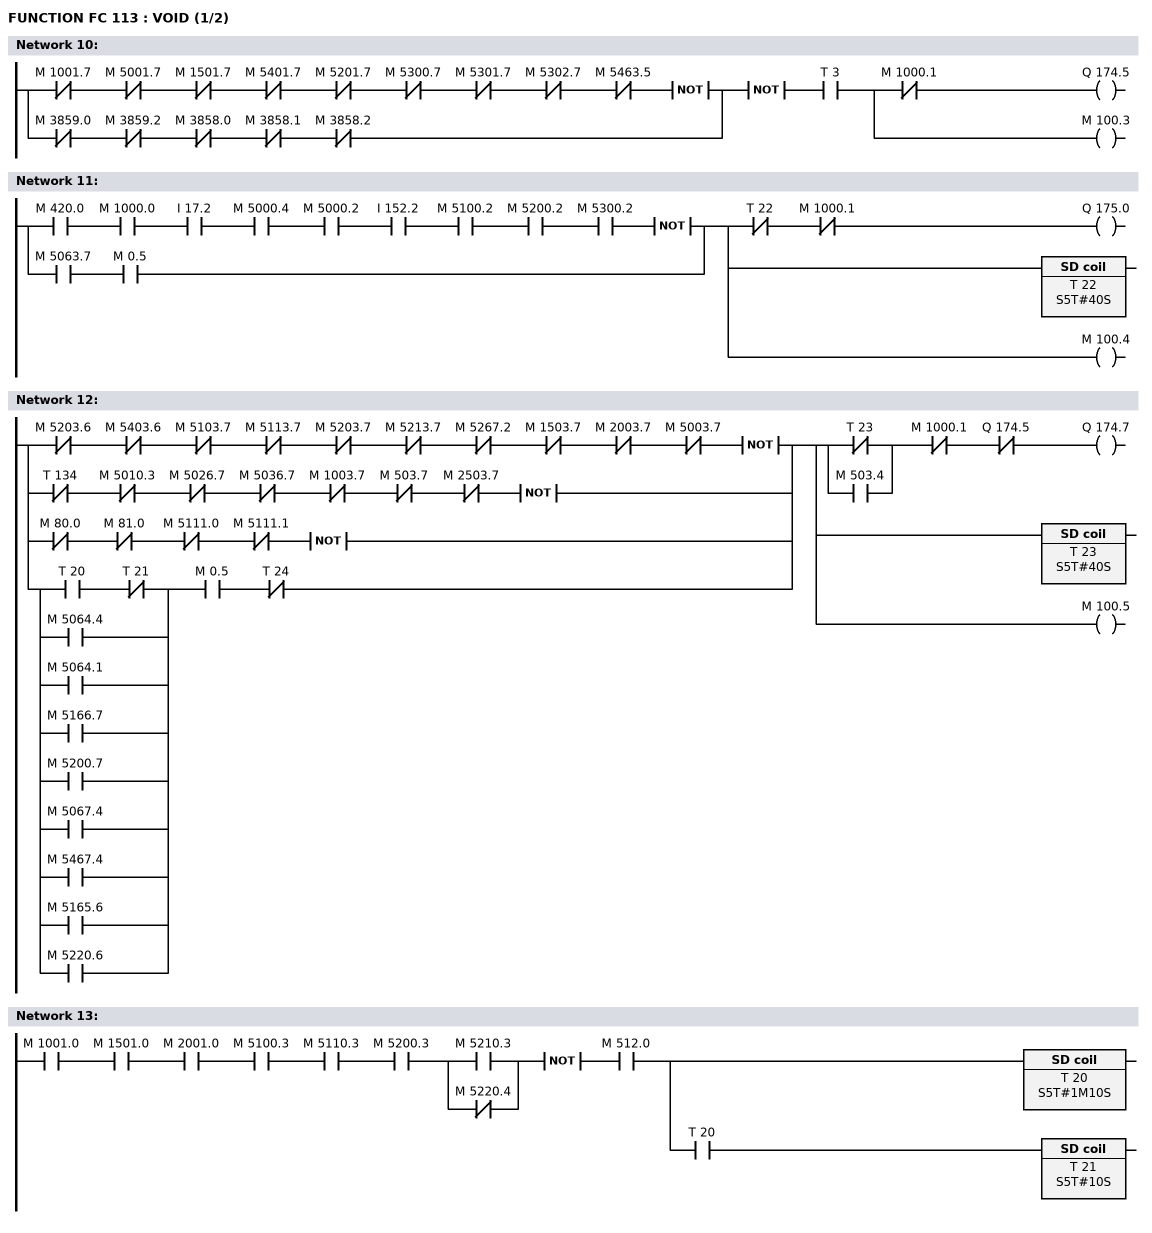

      AN    M   1001.7;
      AN    M   5001.7;
      AN    M   1501.7;
      AN    M   5401.7;
      AN    M   5201.7;
      AN    M   5300.7;
      AN    M   5301.7;
      AN    M   5302.7;
      AN    M   5463.5;
      NOT   ;
      O     ;
      AN    M   3859.0;
      AN    M   3859.2;
      AN    M   3858.0;
      AN    M   3858.1;
      AN    M   3858.2;
      NOT   ;
      A     T      3;
      =     L      0.0;
      A     L      0.0;
      AN    M   1000.1;
      =     Q    174.5;
      A     L      0.0;
      BLD   102;
      =     M    100.3;
NETWORK
TITLE =

      A     M    420.0;
      A     M   1000.0;
      A     I     17.2;
      A     M   5000.4;
      A     M   5000.2;
      A     I    152.2;
      A     M   5100.2;
      A     M   5200.2;
      A     M   5300.2;
      NOT   ;
      O     ;
      A     M   5063.7;
      A     M      0.5;
      =     L      0.0;
      A     L      0.0;
      AN    T     22;
      AN    M   1000.1;
      =     Q    175.0;
      A     L      0.0;
      BLD   102;
      L     S5T#40S;
      SD    T     22;
      A     L      0.0;
      BLD   102;
      =     M    100.4;
NETWORK
TITLE =

      AN    M   5203.6;
      AN    M   5403.6;
      AN    M   5103.7;
      AN    M   5113.7;
      AN    M   5203.7;
      AN    M   5213.7;
      AN    M   5267.2;
      AN    M   1503.7;
      AN    M   2003.7;
      AN    M   5003.7;
      NOT   ;
      O(    ;
      AN    T    134;
      AN    M   5010.3;
      AN    M   5026.7;
      AN    M   5036.7;
      AN    M   1003.7;
      AN    M    503.7;
      AN    M   2503.7;
      NOT   ;
      )     ;
      O(    ;
      AN    M     80.0;
      AN    M     81.0;
      AN    M   5111.0;
      AN    M   5111.1;
      NOT   ;
      )     ;
      O     ;
      A(    ;
      A     T     20;
      AN    T     21;
      O     M   5064.4;
      O     M   5064.1;
      O     M   5166.7;
      O     M   5200.7;
      O     M   5067.4;
      O     M   5467.4;
      O     M   5165.6;
      O     M   5220.6;
      )     ;
      A     M      0.5;
      AN    T     24;
      =     L      0.0;
      A     L      0.0;
      A(    ;
      ON    T     23;
      O     M    503.4;
      )     ;
      AN    M   1000.1;
      AN    Q    174.5;
      =     Q    174.7;
      A     L      0.0;
      BLD   102;
      L     S5T#40S;
      SD    T     23;
      A     L      0.0;
      BLD   102;
      =     M    100.5;
NETWORK
TITLE =

      A     M   1001.0;
      A     M   1501.0;
      A     M   2001.0;
      A     M   5100.3;
      A     M   5110.3;
      A     M   5200.3;
      A(    ;
      O     M   5210.3;
      ON    M   5220.4;
      )     ;
      NOT   ;
      A     M    512.0;
      =     L      0.0;
      A     L      0.0;
      BLD   102;
      L     S5T#1M10S;
      SD    T     20;
      A     L      0.0;
      A     T     20;
      L     S5T#10S;
      SD    T     21;
NETWORK
TITLE =
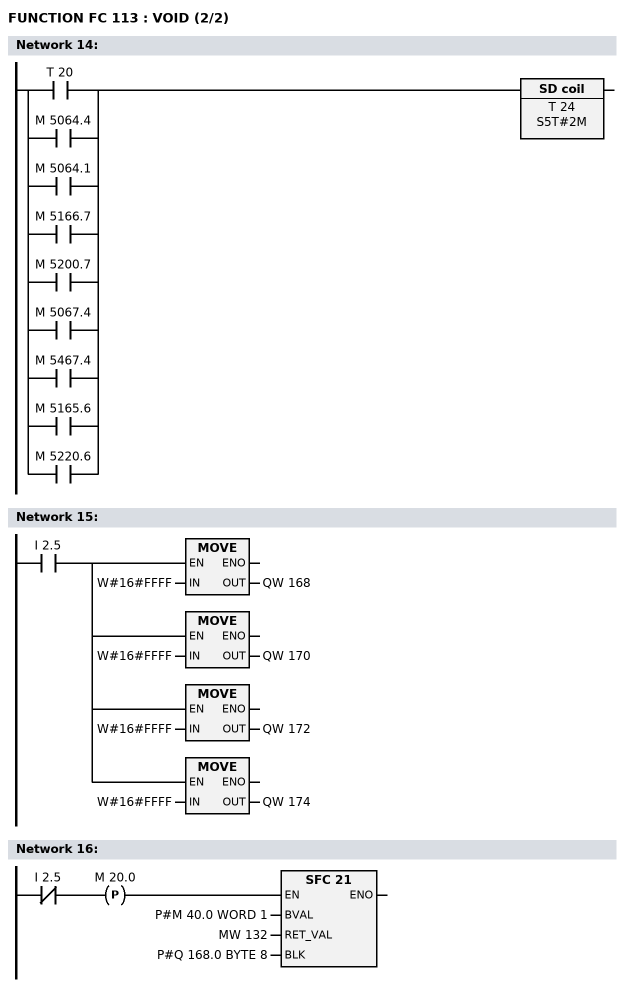

      O     T     20;
      O     M   5064.4;
      O     M   5064.1;
      O     M   5166.7;
      O     M   5200.7;
      O     M   5067.4;
      O     M   5467.4;
      O     M   5165.6;
      O     M   5220.6;
      L     S5T#2M;
      SD    T     24;
NETWORK
TITLE =

      A     I      2.5;
      =     L      0.0;
      A     L      0.0;
      JNB   _003;
      L     W#16#FFFF;
      T     QW   168;
_003: NOP   0;
      A     L      0.0;
      JNB   _004;
      L     W#16#FFFF;
      T     QW   170;
_004: NOP   0;
      A     L      0.0;
      JNB   _005;
      L     W#16#FFFF;
      T     QW   172;
_005: NOP   0;
      A     L      0.0;
      JNB   _006;
      L     W#16#FFFF;
      T     QW   174;
_006: NOP   0;
NETWORK
TITLE =

      AN    I      2.5;
      FP    M     20.0;
      JNB   _007;
      CALL SFC   21 (
           BVAL                     := P#M 40.0 WORD 1,
           RET_VAL                  := MW   132,
           BLK                      := P#Q 168.0 BYTE 8);
_007: NOP   0;
END_FUNCTION

FUNCTION_BLOCK FB 120
TITLE =
VERSION : 0.1


VAR
  S702_MODE : FB 402;
END_VAR
BEGIN
NETWORK
TITLE =
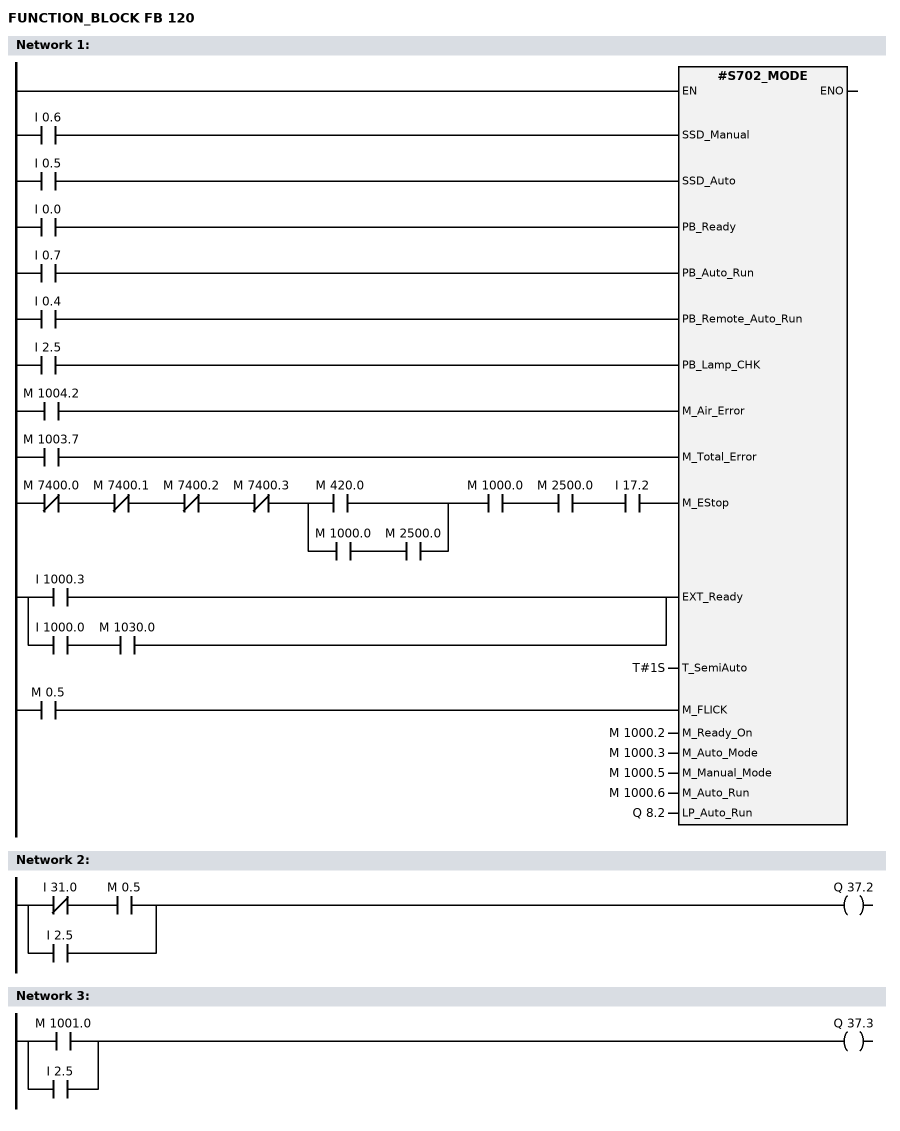

      A     I      0.6;
      =     L      0.0;
      BLD   103;
      A     I      0.5;
      =     L      0.1;
      BLD   103;
      A     I      0.0;
      =     L      0.2;
      BLD   103;
      A     I      0.7;
      =     L      0.3;
      BLD   103;
      A     I      0.4;
      =     L      0.5;
      BLD   103;
      A     I      2.5;
      =     L      0.6;
      BLD   103;
      A     M   1004.2;
      =     L      0.7;
      BLD   103;
      A     M   1003.7;
      =     L      1.1;
      BLD   103;
      AN    M   7400.0;
      AN    M   7400.1;
      AN    M   7400.2;
      AN    M   7400.3;
      A(    ;
      O     M    420.0;
      O     ;
      A     M   1000.0;
      A     M   2500.0;
      )     ;
      A     M   1000.0;
      A     M   2500.0;
      A     I     17.2;
      =     L      1.2;
      BLD   103;
      A(    ;
      O     I   1000.3;
      O     ;
      A     I   1000.0;
      A     M   1030.0;
      )     ;
      =     L      1.3;
      BLD   103;
      A     M      0.5;
      =     L      1.5;
      BLD   103;
      CALL #S702_MODE (
           SSD_Manual               := L      0.0,
           SSD_Auto                 := L      0.1,
           PB_Ready                 := L      0.2,
           PB_Auto_Run              := L      0.3,
           PB_Remote_Auto_Run       := L      0.5,
           PB_Lamp_CHK              := L      0.6,
           M_Air_Error              := L      0.7,
           M_Total_Error            := L      1.1,
           M_EStop                  := L      1.2,
           EXT_Ready                := L      1.3,
           T_SemiAuto               := T#1S,
           M_FLICK                  := L      1.5,
           M_Ready_On               := M   1000.2,
           M_Auto_Mode              := M   1000.3,
           M_Manual_Mode            := M   1000.5,
           M_Auto_Run               := M   1000.6,
           LP_Auto_Run              := Q      8.2);
      NOP   0;
NETWORK
TITLE =

      AN    I     31.0;
      A     M      0.5;
      O     I      2.5;
      =     Q     37.2;
NETWORK
TITLE =

      O     M   1001.0;
      O     I      2.5;
      =     Q     37.3;
END_FUNCTION_BLOCK

DATA_BLOCK DB 120
TITLE =
VERSION : 0.0

 FB 120
BEGIN
   S702_MODE.SSD_Manual := FALSE;
   S702_MODE.SSD_Auto := FALSE;
   S702_MODE.PB_Ready := FALSE;
   S702_MODE.PB_Auto_Run := FALSE;
   S702_MODE.PB_Remote_Ready := FALSE;
   S702_MODE.PB_Remote_Auto_Run := FALSE;
   S702_MODE.PB_Lamp_CHK := FALSE;
   S702_MODE.M_Air_Error := FALSE;
   S702_MODE.M_Water_Error := FALSE;
   S702_MODE.M_Total_Error := FALSE;
   S702_MODE.M_EStop := FALSE;
   S702_MODE.EXT_Ready := FALSE;
   S702_MODE.EXT_Auto := FALSE;
   S702_MODE.T_SemiAuto := T#0MS;
   S702_MODE.M_FLICK := FALSE;
   S702_MODE.M_Ready_On := FALSE;
   S702_MODE.M_Auto_Mode := FALSE;
   S702_MODE.M_SemiAuto_Mode := FALSE;
   S702_MODE.M_Manual_Mode := FALSE;
   S702_MODE.M_Auto_Run := FALSE;
   S702_MODE.LP_Ready_On := FALSE;
   S702_MODE.LP_Auto_Run := FALSE;
   S702_MODE.AUTO_MODE_DELAY.IN := FALSE;
   S702_MODE.AUTO_MODE_DELAY.PT := T#0MS;
   S702_MODE.AUTO_MODE_DELAY.Q := FALSE;
   S702_MODE.AUTO_MODE_DELAY.ET := T#0MS;
   S702_MODE.AUTO_MODE_DELAY.STATE := B#16#0;
   S702_MODE.AUTO_MODE_DELAY.STIME := T#0MS;
   S702_MODE.AUTO_MODE_DELAY.ATIME := T#0MS;
   S702_MODE.SEMI_AUTO_DELAY.IN := FALSE;
   S702_MODE.SEMI_AUTO_DELAY.PT := T#0MS;
   S702_MODE.SEMI_AUTO_DELAY.Q := FALSE;
   S702_MODE.SEMI_AUTO_DELAY.ET := T#0MS;
   S702_MODE.SEMI_AUTO_DELAY.STATE := B#16#0;
   S702_MODE.SEMI_AUTO_DELAY.STIME := T#0MS;
   S702_MODE.SEMI_AUTO_DELAY.ATIME := T#0MS;
   S702_MODE.MANUAL_DELAY.IN := FALSE;
   S702_MODE.MANUAL_DELAY.PT := T#0MS;
   S702_MODE.MANUAL_DELAY.Q := FALSE;
   S702_MODE.MANUAL_DELAY.ET := T#0MS;
   S702_MODE.MANUAL_DELAY.STATE := B#16#0;
   S702_MODE.MANUAL_DELAY.STIME := T#0MS;
   S702_MODE.MANUAL_DELAY.ATIME := T#0MS;
END_DATA_BLOCK

FUNCTION FC 120 : VOID
TITLE =
VERSION : 0.1

BEGIN
NETWORK
TITLE =
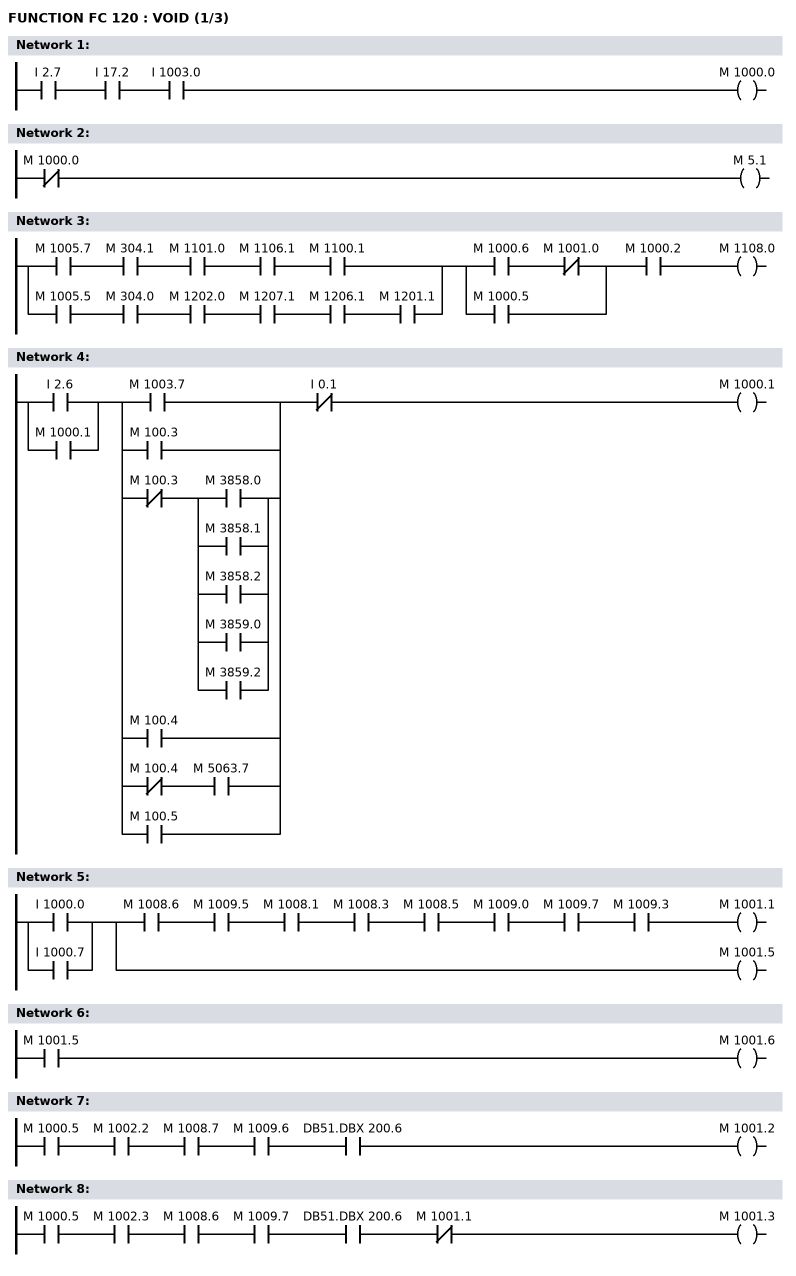

      A     I      2.7;
      A     I     17.2;
      A     I   1003.0;
      =     M   1000.0;
NETWORK
TITLE =

      AN    M   1000.0;
      =     M      5.1;
NETWORK
TITLE =

      A(    ;
      A     M   1005.7;
      A     M    304.1;
      A     M   1101.0;
      A     M   1106.1;
      A     M   1100.1;
      O     ;
      A     M   1005.5;
      A     M    304.0;
      A     M   1202.0;
      A     M   1207.1;
      A     M   1206.1;
      A     M   1201.1;
      )     ;
      A(    ;
      A     M   1000.6;
      AN    M   1001.0;
      O     M   1000.5;
      )     ;
      A     M   1000.2;
      =     M   1108.0;
NETWORK
TITLE =

      A(    ;
      O     I      2.6;
      O     M   1000.1;
      )     ;
      A(    ;
      O     M   1003.7;
      O     M    100.3;
      O     ;
      AN    M    100.3;
      A(    ;
      O     M   3858.0;
      O     M   3858.1;
      O     M   3858.2;
      O     M   3859.0;
      O     M   3859.2;
      )     ;
      O     M    100.4;
      O     ;
      AN    M    100.4;
      A     M   5063.7;
      O     M    100.5;
      )     ;
      AN    I      0.1;
      =     M   1000.1;
NETWORK
TITLE =

      O     I   1000.0;
      O     I   1000.7;
      =     L      0.0;
      A     L      0.0;
      A     M   1008.6;
      A     M   1009.5;
      A     M   1008.1;
      A     M   1008.3;
      A     M   1008.5;
      A     M   1009.0;
      A     M   1009.7;
      A     M   1009.3;
      =     M   1001.1;
      A     L      0.0;
      BLD   102;
      =     M   1001.5;
NETWORK
TITLE =

      A     M   1001.5;
      =     M   1001.6;
NETWORK
TITLE =

      A     M   1000.5;
      A     M   1002.2;
      A     M   1008.7;
      A     M   1009.6;
      A     DB51.DBX  200.6;
      =     M   1001.2;
NETWORK
TITLE =

      A     M   1000.5;
      A     M   1002.3;
      A     M   1008.6;
      A     M   1009.7;
      A     DB51.DBX  200.6;
      AN    M   1001.1;
      =     M   1001.3;
NETWORK
TITLE =
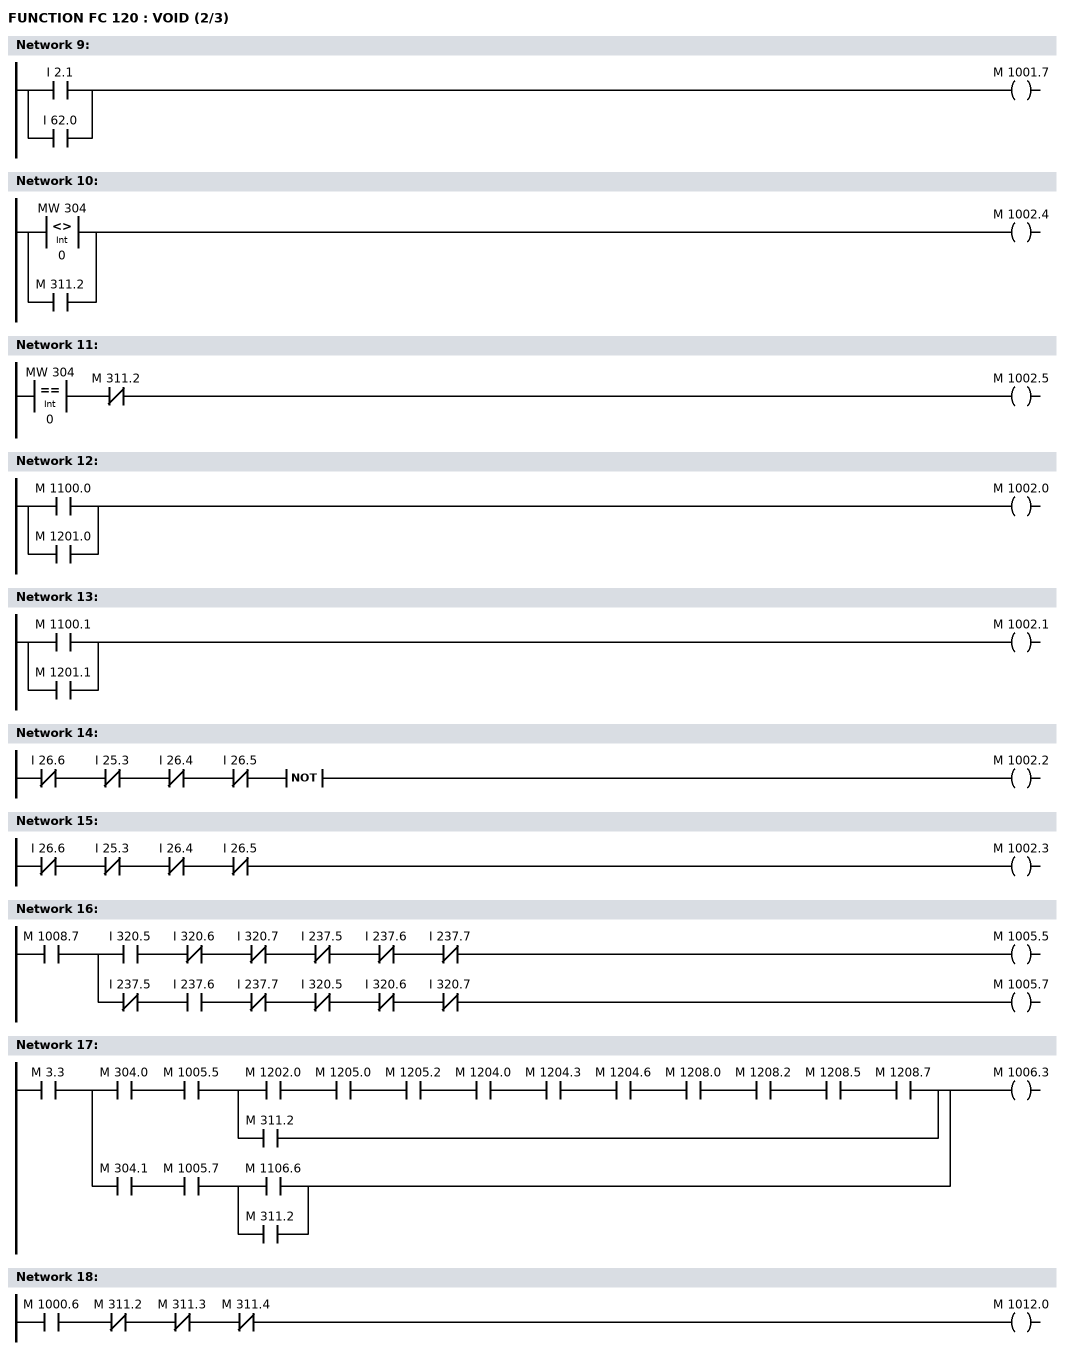

      O     I      2.1;
      O     I     62.0;
      =     M   1001.7;
NETWORK
TITLE =

      O(    ;
      L     MW   304;
      L     0;
      <>I   ;
      )     ;
      O     M    311.2;
      =     M   1002.4;
NETWORK
TITLE =

      A(    ;
      L     MW   304;
      L     0;
      ==I   ;
      )     ;
      AN    M    311.2;
      =     M   1002.5;
NETWORK
TITLE =

      O     M   1100.0;
      O     M   1201.0;
      =     M   1002.0;
NETWORK
TITLE =

      O     M   1100.1;
      O     M   1201.1;
      =     M   1002.1;
NETWORK
TITLE =

      AN    I     26.6;
      AN    I     25.3;
      AN    I     26.4;
      AN    I     26.5;
      NOT   ;
      =     M   1002.2;
NETWORK
TITLE =

      AN    I     26.6;
      AN    I     25.3;
      AN    I     26.4;
      AN    I     26.5;
      =     M   1002.3;
NETWORK
TITLE =

      A     M   1008.7;
      =     L      0.0;
      A     L      0.0;
      A     I    320.5;
      AN    I    320.6;
      AN    I    320.7;
      AN    I    237.5;
      AN    I    237.6;
      AN    I    237.7;
      =     M   1005.5;
      A     L      0.0;
      AN    I    237.5;
      A     I    237.6;
      AN    I    237.7;
      AN    I    320.5;
      AN    I    320.6;
      AN    I    320.7;
      =     M   1005.7;
NETWORK
TITLE =

      A     M      3.3;
      A(    ;
      A     M    304.0;
      A     M   1005.5;
      A(    ;
      A     M   1202.0;
      A     M   1205.0;
      A     M   1205.2;
      A     M   1204.0;
      A     M   1204.3;
      A     M   1204.6;
      A     M   1208.0;
      A     M   1208.2;
      A     M   1208.5;
      A     M   1208.7;
      O     M    311.2;
      )     ;
      O     ;
      A     M    304.1;
      A     M   1005.7;
      A(    ;
      O     M   1106.6;
      O     M    311.2;
      )     ;
      )     ;
      =     M   1006.3;
NETWORK
TITLE =

      A     M   1000.6;
      AN    M    311.2;
      AN    M    311.3;
      AN    M    311.4;
      =     M   1012.0;
NETWORK
TITLE =
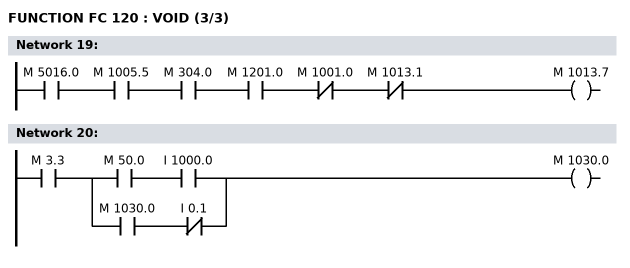

      A     M   5016.0;
      A     M   1005.5;
      A     M    304.0;
      A     M   1201.0;
      AN    M   1001.0;
      AN    M   1013.1;
      =     M   1013.7;
NETWORK
TITLE =

      A     M      3.3;
      A(    ;
      A     M     50.0;
      A     I   1000.0;
      O     ;
      A     M   1030.0;
      AN    I      0.1;
      )     ;
      =     M   1030.0;
NETWORK
TITLE =

      AN    OV;
      =     L      0.0;
      A(    ;
      A(    ;
      A     L      0.0;
      AN    M   1005.7;
      JNB   _001;
      L     0;
      T     MW  1150;
      SET   ;
      SAVE  ;
      CLR   ;
_001: A     BR;
      )     ;
      JNB   _002;
      L     0;
      T     MW  1152;
      SET   ;
      SAVE  ;
      CLR   ;
_002: A     BR;
      )     ;
      JNB   _003;
      L     0;
      T     MB  1154;
_003: NOP   0;
      A(    ;
      A(    ;
      A     L      0.0;
      AN    M   1005.5;
      JNB   _004;
      L     0;
      T     MW  1250;
      SET   ;
      SAVE  ;
      CLR   ;
_004: A     BR;
      )     ;
      JNB   _005;
      L     0;
      T     MW  1252;
      SET   ;
      SAVE  ;
      CLR   ;
_005: A     BR;
      )     ;
      JNB   _006;
      L     0;
      T     MB  1254;
_006: NOP   0;
NETWORK
TITLE =

      AN    M   1007.4;
      =     L      0.0;
      A     L      0.0;
      JNB   _007;
      CALL SFC   21 (
           BVAL                     := P#M 40.0 WORD 1,
           RET_VAL                  := MW   132,
           BLK                      := P#M 1100.0 BYTE 10);
_007: NOP   0;
      A     L      0.0;
      JNB   _008;
      CALL SFC   21 (
           BVAL                     := P#M 40.0 WORD 1,
           RET_VAL                  := MW   132,
           BLK                      := P#Q 236.0 BYTE 4);
_008: NOP   0;
      A     L      0.0;
      JNB   _009;
      CALL SFC   21 (
           BVAL                     := P#M 40.0 WORD 1,
           RET_VAL                  := MW   132,
           BLK                      := P#M 1200.0 BYTE 12);
_009: NOP   0;
      A     L      0.0;
      JNB   _00a;
      CALL SFC   21 (
           BVAL                     := P#M 40.0 WORD 1,
           RET_VAL                  := MW   132,
           BLK                      := P#M 1240.0 BYTE 5);
_00a: NOP   0;
      A     L      0.0;
      JNB   _00b;
      CALL SFC   21 (
           BVAL                     := P#M 40.0 WORD 1,
           RET_VAL                  := MW   132,
           BLK                      := P#Q 332.0 BYTE 6);
_00b: NOP   0;
END_FUNCTION

FUNCTION_BLOCK FB 121
TITLE =
VERSION : 0.1


VAR
  S702_HOOK_PIN : FB 424;
  S702_DAECHA_LOCK : FB 424;
  S702_DAECHA_LOCK_UP_DN : FB 424;
  S702_ELE : FB 424;
  S702_AIR_ELE : FB 424;
  S702_EJECT : FB 424;
  S702_DAECHA_STOPPER : FB 424;
  S702_DAECHA_CLAMP : FB 424;
  S702_SHOCK_ABSORBER : FB 424;
END_VAR
BEGIN
NETWORK
TITLE =
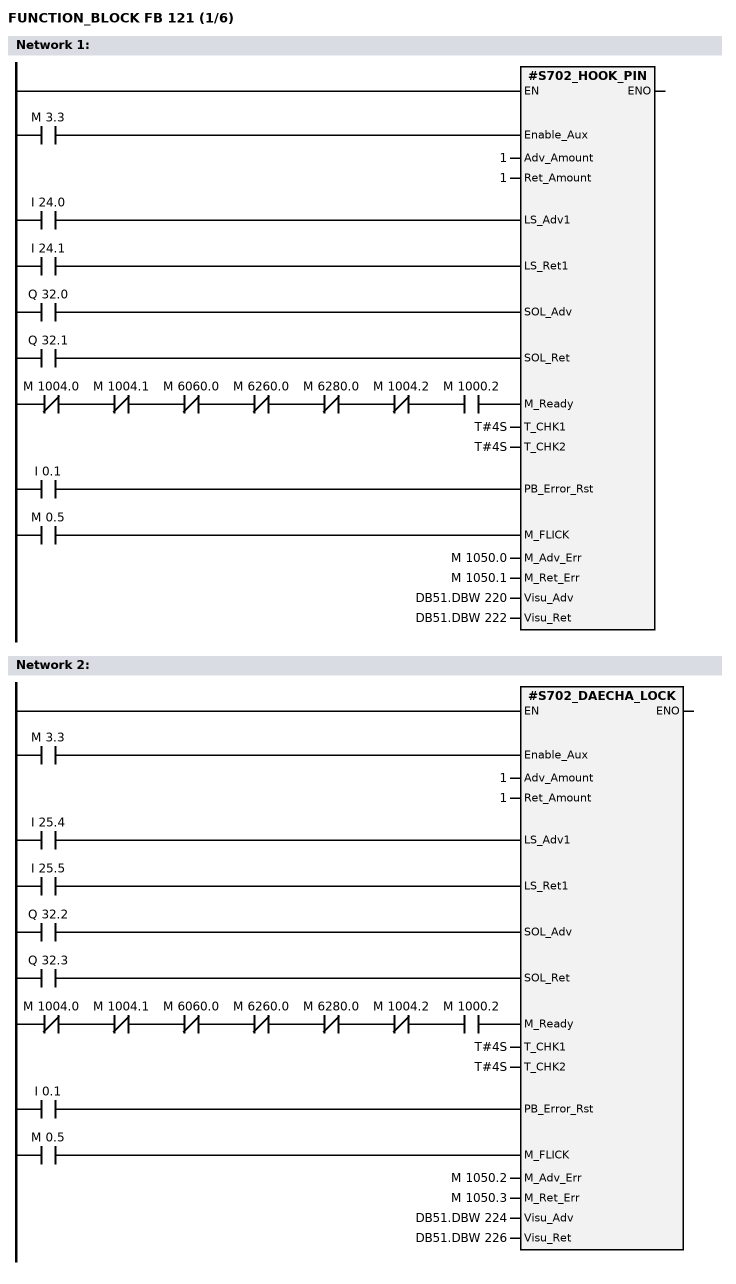

      A     M      3.3;
      =     L      0.0;
      BLD   103;
      A     I     24.0;
      =     L      0.1;
      BLD   103;
      A     I     24.1;
      =     L      0.2;
      BLD   103;
      A     Q     32.0;
      =     L      1.1;
      BLD   103;
      A     Q     32.1;
      =     L      1.2;
      BLD   103;
      AN    M   1004.0;
      AN    M   1004.1;
      AN    M   6060.0;
      AN    M   6260.0;
      AN    M   6280.0;
      AN    M   1004.2;
      A     M   1000.2;
      =     L      1.3;
      BLD   103;
      A     I      0.1;
      =     L      1.5;
      BLD   103;
      A     M      0.5;
      =     L      1.6;
      BLD   103;
      CALL #S702_HOOK_PIN (
           Enable_Aux               := L      0.0,
           Adv_Amount               := 1,
           Ret_Amount               := 1,
           LS_Adv1                  := L      0.1,
           LS_Ret1                  := L      0.2,
           SOL_Adv                  := L      1.1,
           SOL_Ret                  := L      1.2,
           M_Ready                  := L      1.3,
           T_CHK1                   := T#4S,
           T_CHK2                   := T#4S,
           PB_Error_Rst             := L      1.5,
           M_FLICK                  := L      1.6,
           M_Adv_Err                := M   1050.0,
           M_Ret_Err                := M   1050.1,
           Visu_Adv                 := DB51.DBW  220,
           Visu_Ret                 := DB51.DBW  222);
      NOP   0;
NETWORK
TITLE =

      A     M      3.3;
      =     L      0.0;
      BLD   103;
      A     I     25.4;
      =     L      0.1;
      BLD   103;
      A     I     25.5;
      =     L      0.2;
      BLD   103;
      A     Q     32.2;
      =     L      1.1;
      BLD   103;
      A     Q     32.3;
      =     L      1.2;
      BLD   103;
      AN    M   1004.0;
      AN    M   1004.1;
      AN    M   6060.0;
      AN    M   6260.0;
      AN    M   6280.0;
      AN    M   1004.2;
      A     M   1000.2;
      =     L      1.3;
      BLD   103;
      A     I      0.1;
      =     L      1.5;
      BLD   103;
      A     M      0.5;
      =     L      1.6;
      BLD   103;
      CALL #S702_DAECHA_LOCK (
           Enable_Aux               := L      0.0,
           Adv_Amount               := 1,
           Ret_Amount               := 1,
           LS_Adv1                  := L      0.1,
           LS_Ret1                  := L      0.2,
           SOL_Adv                  := L      1.1,
           SOL_Ret                  := L      1.2,
           M_Ready                  := L      1.3,
           T_CHK1                   := T#4S,
           T_CHK2                   := T#4S,
           PB_Error_Rst             := L      1.5,
           M_FLICK                  := L      1.6,
           M_Adv_Err                := M   1050.2,
           M_Ret_Err                := M   1050.3,
           Visu_Adv                 := DB51.DBW  224,
           Visu_Ret                 := DB51.DBW  226);
      NOP   0;
NETWORK
TITLE =
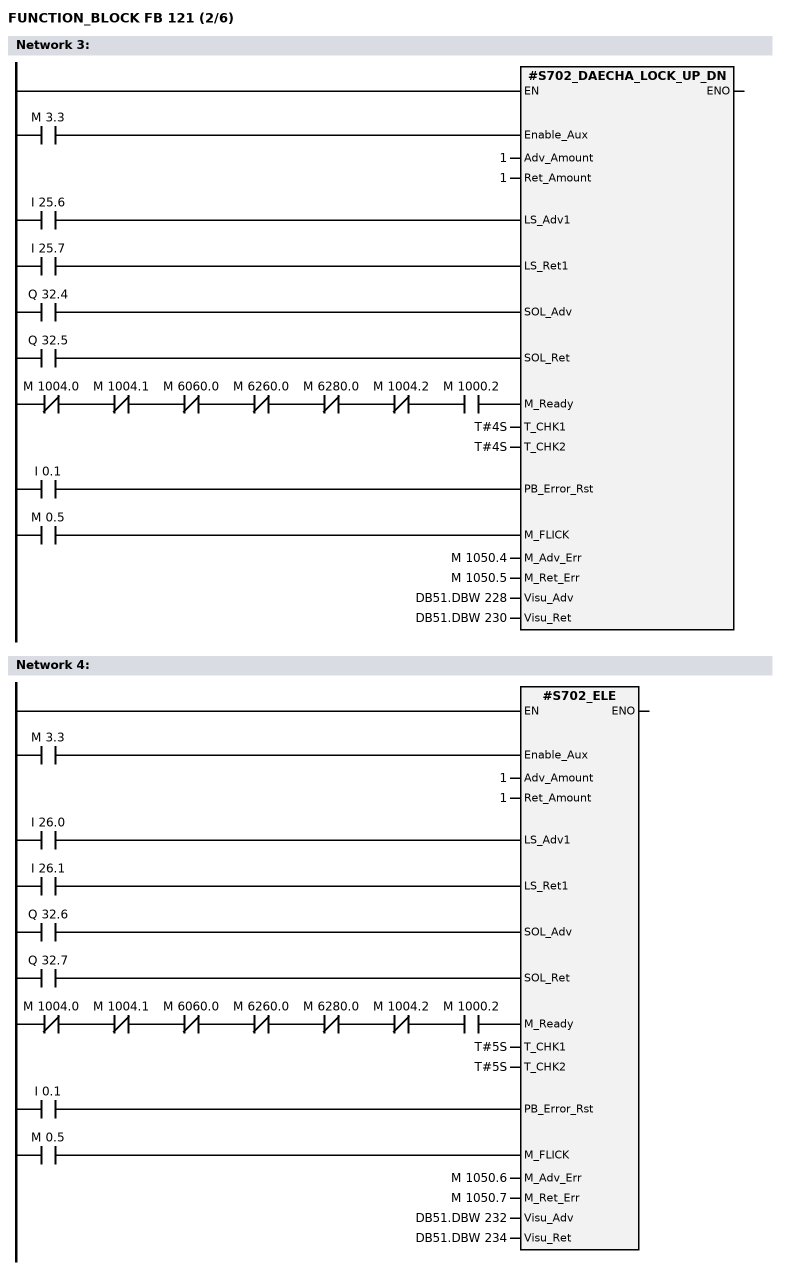

      A     M      3.3;
      =     L      0.0;
      BLD   103;
      A     I     25.6;
      =     L      0.1;
      BLD   103;
      A     I     25.7;
      =     L      0.2;
      BLD   103;
      A     Q     32.4;
      =     L      1.1;
      BLD   103;
      A     Q     32.5;
      =     L      1.2;
      BLD   103;
      AN    M   1004.0;
      AN    M   1004.1;
      AN    M   6060.0;
      AN    M   6260.0;
      AN    M   6280.0;
      AN    M   1004.2;
      A     M   1000.2;
      =     L      1.3;
      BLD   103;
      A     I      0.1;
      =     L      1.5;
      BLD   103;
      A     M      0.5;
      =     L      1.6;
      BLD   103;
      CALL #S702_DAECHA_LOCK_UP_DN (
           Enable_Aux               := L      0.0,
           Adv_Amount               := 1,
           Ret_Amount               := 1,
           LS_Adv1                  := L      0.1,
           LS_Ret1                  := L      0.2,
           SOL_Adv                  := L      1.1,
           SOL_Ret                  := L      1.2,
           M_Ready                  := L      1.3,
           T_CHK1                   := T#4S,
           T_CHK2                   := T#4S,
           PB_Error_Rst             := L      1.5,
           M_FLICK                  := L      1.6,
           M_Adv_Err                := M   1050.4,
           M_Ret_Err                := M   1050.5,
           Visu_Adv                 := DB51.DBW  228,
           Visu_Ret                 := DB51.DBW  230);
      NOP   0;
NETWORK
TITLE =

      A     M      3.3;
      =     L      0.0;
      BLD   103;
      A     I     26.0;
      =     L      0.1;
      BLD   103;
      A     I     26.1;
      =     L      0.2;
      BLD   103;
      A     Q     32.6;
      =     L      1.1;
      BLD   103;
      A     Q     32.7;
      =     L      1.2;
      BLD   103;
      AN    M   1004.0;
      AN    M   1004.1;
      AN    M   6060.0;
      AN    M   6260.0;
      AN    M   6280.0;
      AN    M   1004.2;
      A     M   1000.2;
      =     L      1.3;
      BLD   103;
      A     I      0.1;
      =     L      1.5;
      BLD   103;
      A     M      0.5;
      =     L      1.6;
      BLD   103;
      CALL #S702_ELE (
           Enable_Aux               := L      0.0,
           Adv_Amount               := 1,
           Ret_Amount               := 1,
           LS_Adv1                  := L      0.1,
           LS_Ret1                  := L      0.2,
           SOL_Adv                  := L      1.1,
           SOL_Ret                  := L      1.2,
           M_Ready                  := L      1.3,
           T_CHK1                   := T#5S,
           T_CHK2                   := T#5S,
           PB_Error_Rst             := L      1.5,
           M_FLICK                  := L      1.6,
           M_Adv_Err                := M   1050.6,
           M_Ret_Err                := M   1050.7,
           Visu_Adv                 := DB51.DBW  232,
           Visu_Ret                 := DB51.DBW  234);
      NOP   0;
NETWORK
TITLE =
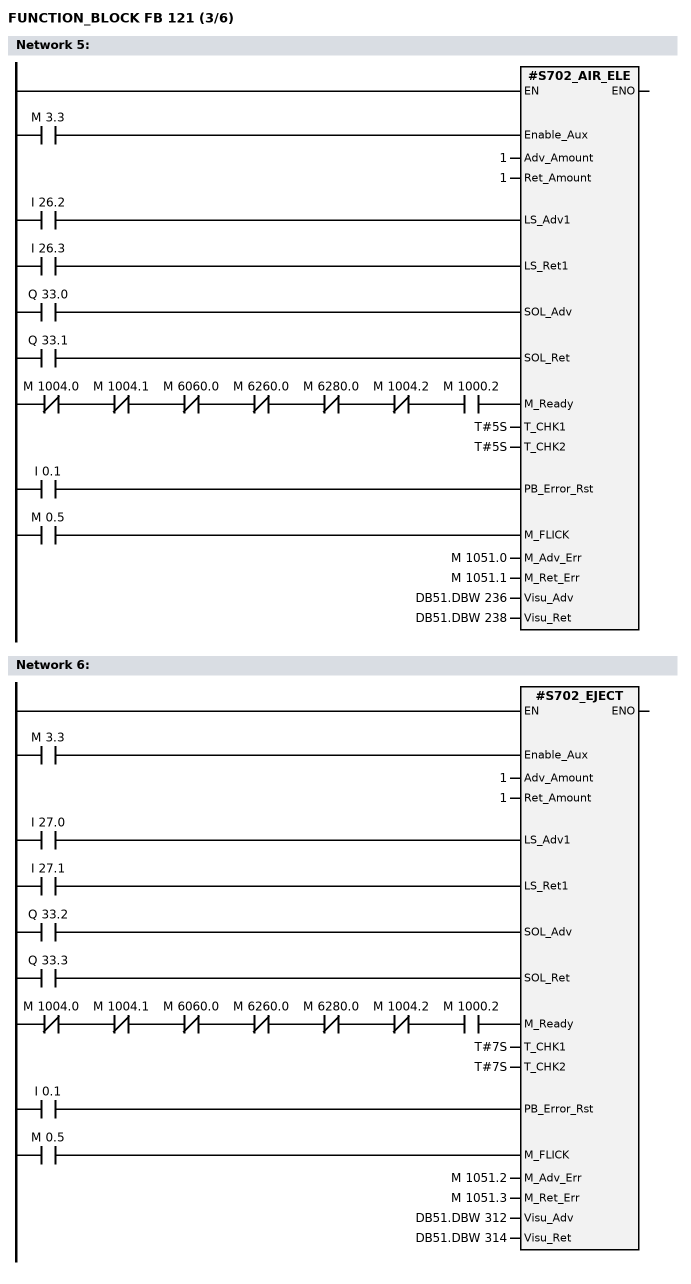

      A     M      3.3;
      =     L      0.0;
      BLD   103;
      A     I     26.2;
      =     L      0.1;
      BLD   103;
      A     I     26.3;
      =     L      0.2;
      BLD   103;
      A     Q     33.0;
      =     L      1.1;
      BLD   103;
      A     Q     33.1;
      =     L      1.2;
      BLD   103;
      AN    M   1004.0;
      AN    M   1004.1;
      AN    M   6060.0;
      AN    M   6260.0;
      AN    M   6280.0;
      AN    M   1004.2;
      A     M   1000.2;
      =     L      1.3;
      BLD   103;
      A     I      0.1;
      =     L      1.5;
      BLD   103;
      A     M      0.5;
      =     L      1.6;
      BLD   103;
      CALL #S702_AIR_ELE (
           Enable_Aux               := L      0.0,
           Adv_Amount               := 1,
           Ret_Amount               := 1,
           LS_Adv1                  := L      0.1,
           LS_Ret1                  := L      0.2,
           SOL_Adv                  := L      1.1,
           SOL_Ret                  := L      1.2,
           M_Ready                  := L      1.3,
           T_CHK1                   := T#5S,
           T_CHK2                   := T#5S,
           PB_Error_Rst             := L      1.5,
           M_FLICK                  := L      1.6,
           M_Adv_Err                := M   1051.0,
           M_Ret_Err                := M   1051.1,
           Visu_Adv                 := DB51.DBW  236,
           Visu_Ret                 := DB51.DBW  238);
      NOP   0;
NETWORK
TITLE =

      A     M      3.3;
      =     L      0.0;
      BLD   103;
      A     I     27.0;
      =     L      0.1;
      BLD   103;
      A     I     27.1;
      =     L      0.2;
      BLD   103;
      A     Q     33.2;
      =     L      1.1;
      BLD   103;
      A     Q     33.3;
      =     L      1.2;
      BLD   103;
      AN    M   1004.0;
      AN    M   1004.1;
      AN    M   6060.0;
      AN    M   6260.0;
      AN    M   6280.0;
      AN    M   1004.2;
      A     M   1000.2;
      =     L      1.3;
      BLD   103;
      A     I      0.1;
      =     L      1.5;
      BLD   103;
      A     M      0.5;
      =     L      1.6;
      BLD   103;
      CALL #S702_EJECT (
           Enable_Aux               := L      0.0,
           Adv_Amount               := 1,
           Ret_Amount               := 1,
           LS_Adv1                  := L      0.1,
           LS_Ret1                  := L      0.2,
           SOL_Adv                  := L      1.1,
           SOL_Ret                  := L      1.2,
           M_Ready                  := L      1.3,
           T_CHK1                   := T#7S,
           T_CHK2                   := T#7S,
           PB_Error_Rst             := L      1.5,
           M_FLICK                  := L      1.6,
           M_Adv_Err                := M   1051.2,
           M_Ret_Err                := M   1051.3,
           Visu_Adv                 := DB51.DBW  312,
           Visu_Ret                 := DB51.DBW  314);
      NOP   0;
NETWORK
TITLE =
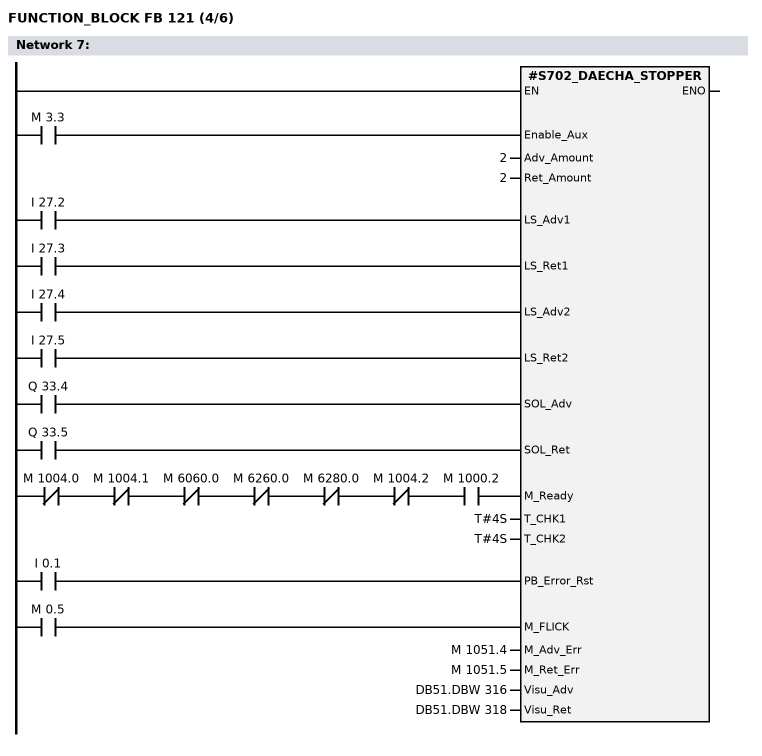

      A     M      3.3;
      =     L      0.0;
      BLD   103;
      A     I     27.2;
      =     L      0.1;
      BLD   103;
      A     I     27.3;
      =     L      0.2;
      BLD   103;
      A     I     27.4;
      =     L      0.3;
      BLD   103;
      A     I     27.5;
      =     L      0.4;
      BLD   103;
      A     Q     33.4;
      =     L      1.1;
      BLD   103;
      A     Q     33.5;
      =     L      1.2;
      BLD   103;
      AN    M   1004.0;
      AN    M   1004.1;
      AN    M   6060.0;
      AN    M   6260.0;
      AN    M   6280.0;
      AN    M   1004.2;
      A     M   1000.2;
      =     L      1.3;
      BLD   103;
      A     I      0.1;
      =     L      1.5;
      BLD   103;
      A     M      0.5;
      =     L      1.6;
      BLD   103;
      CALL #S702_DAECHA_STOPPER (
           Enable_Aux               := L      0.0,
           Adv_Amount               := 2,
           Ret_Amount               := 2,
           LS_Adv1                  := L      0.1,
           LS_Ret1                  := L      0.2,
           LS_Adv2                  := L      0.3,
           LS_Ret2                  := L      0.4,
           SOL_Adv                  := L      1.1,
           SOL_Ret                  := L      1.2,
           M_Ready                  := L      1.3,
           T_CHK1                   := T#4S,
           T_CHK2                   := T#4S,
           PB_Error_Rst             := L      1.5,
           M_FLICK                  := L      1.6,
           M_Adv_Err                := M   1051.4,
           M_Ret_Err                := M   1051.5,
           Visu_Adv                 := DB51.DBW  316,
           Visu_Ret                 := DB51.DBW  318);
      NOP   0;
NETWORK
TITLE =
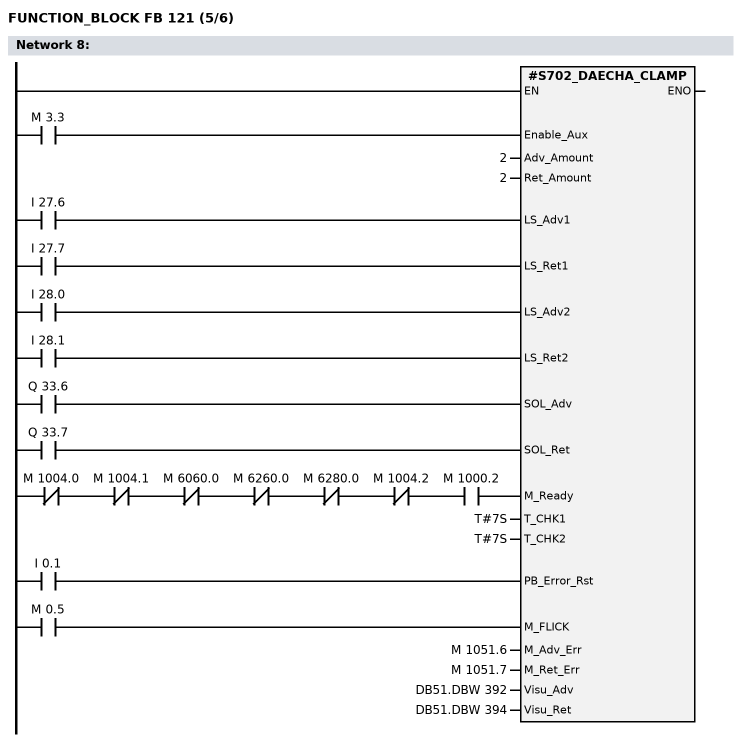

      A     M      3.3;
      =     L      0.0;
      BLD   103;
      A     I     27.6;
      =     L      0.1;
      BLD   103;
      A     I     27.7;
      =     L      0.2;
      BLD   103;
      A     I     28.0;
      =     L      0.3;
      BLD   103;
      A     I     28.1;
      =     L      0.4;
      BLD   103;
      A     Q     33.6;
      =     L      1.1;
      BLD   103;
      A     Q     33.7;
      =     L      1.2;
      BLD   103;
      AN    M   1004.0;
      AN    M   1004.1;
      AN    M   6060.0;
      AN    M   6260.0;
      AN    M   6280.0;
      AN    M   1004.2;
      A     M   1000.2;
      =     L      1.3;
      BLD   103;
      A     I      0.1;
      =     L      1.5;
      BLD   103;
      A     M      0.5;
      =     L      1.6;
      BLD   103;
      CALL #S702_DAECHA_CLAMP (
           Enable_Aux               := L      0.0,
           Adv_Amount               := 2,
           Ret_Amount               := 2,
           LS_Adv1                  := L      0.1,
           LS_Ret1                  := L      0.2,
           LS_Adv2                  := L      0.3,
           LS_Ret2                  := L      0.4,
           SOL_Adv                  := L      1.1,
           SOL_Ret                  := L      1.2,
           M_Ready                  := L      1.3,
           T_CHK1                   := T#7S,
           T_CHK2                   := T#7S,
           PB_Error_Rst             := L      1.5,
           M_FLICK                  := L      1.6,
           M_Adv_Err                := M   1051.6,
           M_Ret_Err                := M   1051.7,
           Visu_Adv                 := DB51.DBW  392,
           Visu_Ret                 := DB51.DBW  394);
      NOP   0;
NETWORK
TITLE =
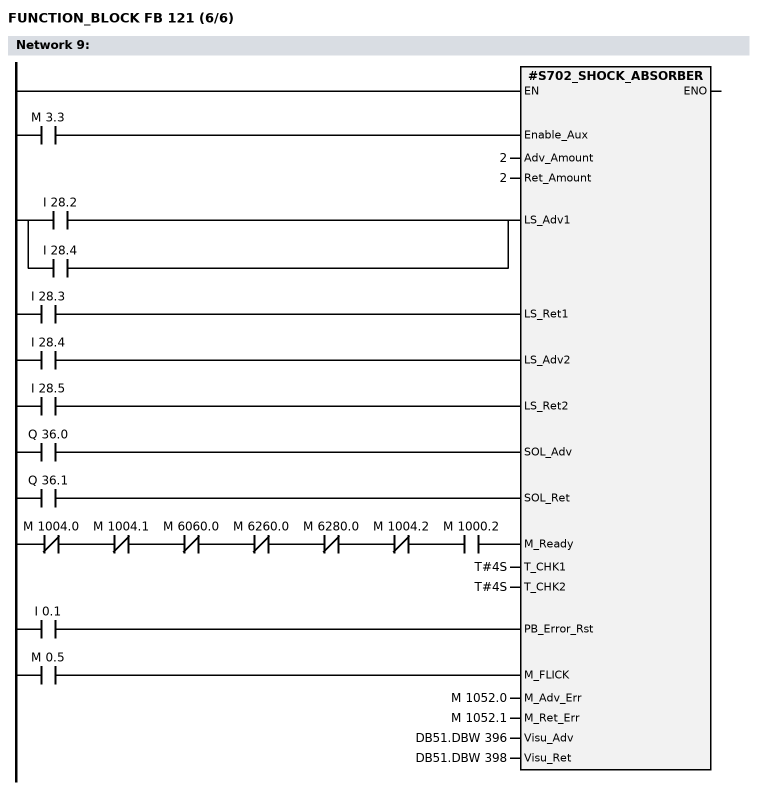

      A     M      3.3;
      =     L      0.0;
      BLD   103;
      A(    ;
      O     I     28.2;
      O     I     28.4;
      )     ;
      =     L      0.1;
      BLD   103;
      A     I     28.3;
      =     L      0.2;
      BLD   103;
      A     I     28.4;
      =     L      0.3;
      BLD   103;
      A     I     28.5;
      =     L      0.4;
      BLD   103;
      A     Q     36.0;
      =     L      1.1;
      BLD   103;
      A     Q     36.1;
      =     L      1.2;
      BLD   103;
      AN    M   1004.0;
      AN    M   1004.1;
      AN    M   6060.0;
      AN    M   6260.0;
      AN    M   6280.0;
      AN    M   1004.2;
      A     M   1000.2;
      =     L      1.3;
      BLD   103;
      A     I      0.1;
      =     L      1.5;
      BLD   103;
      A     M      0.5;
      =     L      1.6;
      BLD   103;
      CALL #S702_SHOCK_ABSORBER (
           Enable_Aux               := L      0.0,
           Adv_Amount               := 2,
           Ret_Amount               := 2,
           LS_Adv1                  := L      0.1,
           LS_Ret1                  := L      0.2,
           LS_Adv2                  := L      0.3,
           LS_Ret2                  := L      0.4,
           SOL_Adv                  := L      1.1,
           SOL_Ret                  := L      1.2,
           M_Ready                  := L      1.3,
           T_CHK1                   := T#4S,
           T_CHK2                   := T#4S,
           PB_Error_Rst             := L      1.5,
           M_FLICK                  := L      1.6,
           M_Adv_Err                := M   1052.0,
           M_Ret_Err                := M   1052.1,
           Visu_Adv                 := DB51.DBW  396,
           Visu_Ret                 := DB51.DBW  398);
      NOP   0;
END_FUNCTION_BLOCK

DATA_BLOCK DB 121
TITLE =
VERSION : 0.0

 FB 121
BEGIN
   S702_HOOK_PIN.Enable_Aux := FALSE;
   S702_HOOK_PIN.Adv_Amount := 0;
   S702_HOOK_PIN.Ret_Amount := 0;
   S702_HOOK_PIN.LS_Adv1 := FALSE;
   S702_HOOK_PIN.LS_Ret1 := FALSE;
   S702_HOOK_PIN.LS_Adv2 := FALSE;
   S702_HOOK_PIN.LS_Ret2 := FALSE;
   S702_HOOK_PIN.LS_Adv3 := FALSE;
   S702_HOOK_PIN.LS_Ret3 := FALSE;
   S702_HOOK_PIN.LS_Adv4 := FALSE;
   S702_HOOK_PIN.LS_Ret4 := FALSE;
   S702_HOOK_PIN.SOL_Adv := FALSE;
   S702_HOOK_PIN.SOL_Ret := FALSE;
   S702_HOOK_PIN.M_Ready := FALSE;
   S702_HOOK_PIN.T_CHK1 := T#0MS;
   S702_HOOK_PIN.T_CHK2 := T#0MS;
   S702_HOOK_PIN.PB_Lamp_CHK := FALSE;
   S702_HOOK_PIN.PB_Error_Rst := FALSE;
   S702_HOOK_PIN.M_FLICK := FALSE;
   S702_HOOK_PIN.M_Adv_Err := FALSE;
   S702_HOOK_PIN.M_Ret_Err := FALSE;
   S702_HOOK_PIN.LP_Adv := FALSE;
   S702_HOOK_PIN.LP_Ret := FALSE;
   S702_HOOK_PIN.Visu_Adv := W#16#0;
   S702_HOOK_PIN.Visu_Ret := W#16#0;
   S702_HOOK_PIN.Error_T1.IN := FALSE;
   S702_HOOK_PIN.Error_T1.PT := T#0MS;
   S702_HOOK_PIN.Error_T1.Q := FALSE;
   S702_HOOK_PIN.Error_T1.ET := T#0MS;
   S702_HOOK_PIN.Error_T1.STATE := B#16#0;
   S702_HOOK_PIN.Error_T1.STIME := T#0MS;
   S702_HOOK_PIN.Error_T1.ATIME := T#0MS;
   S702_HOOK_PIN.Error_T2.IN := FALSE;
   S702_HOOK_PIN.Error_T2.PT := T#0MS;
   S702_HOOK_PIN.Error_T2.Q := FALSE;
   S702_HOOK_PIN.Error_T2.ET := T#0MS;
   S702_HOOK_PIN.Error_T2.STATE := B#16#0;
   S702_HOOK_PIN.Error_T2.STIME := T#0MS;
   S702_HOOK_PIN.Error_T2.ATIME := T#0MS;
   S702_HOOK_PIN.CHK_Aux1 := FALSE;
   S702_HOOK_PIN.CHK_Aux2 := FALSE;
   S702_HOOK_PIN.Error_T1_DN := FALSE;
   S702_HOOK_PIN.Error_T2_DN := FALSE;
   S702_HOOK_PIN.Adv_Memo := FALSE;
   S702_HOOK_PIN.Visu_Adv_Arr[0] := FALSE;
   S702_HOOK_PIN.Visu_Adv_Arr[1] := FALSE;
   S702_HOOK_PIN.Visu_Adv_Arr[2] := FALSE;
   S702_HOOK_PIN.Visu_Adv_Arr[3] := FALSE;
   S702_HOOK_PIN.Visu_Adv_Arr[4] := FALSE;
   S702_HOOK_PIN.Visu_Adv_Arr[5] := FALSE;
   S702_HOOK_PIN.Visu_Adv_Arr[6] := FALSE;
   S702_HOOK_PIN.Visu_Adv_Arr[7] := FALSE;
   S702_HOOK_PIN.Visu_Adv_Arr[8] := FALSE;
   S702_HOOK_PIN.Visu_Adv_Arr[9] := FALSE;
   S702_HOOK_PIN.Visu_Adv_Arr[10] := FALSE;
   S702_HOOK_PIN.Visu_Adv_Arr[11] := FALSE;
   S702_HOOK_PIN.Visu_Adv_Arr[12] := FALSE;
   S702_HOOK_PIN.Visu_Adv_Arr[13] := FALSE;
   S702_HOOK_PIN.Visu_Adv_Arr[14] := FALSE;
   S702_HOOK_PIN.Visu_Adv_Arr[15] := FALSE;
   S702_HOOK_PIN.Visu_Ret_Arr[0] := FALSE;
   S702_HOOK_PIN.Visu_Ret_Arr[1] := FALSE;
   S702_HOOK_PIN.Visu_Ret_Arr[2] := FALSE;
   S702_HOOK_PIN.Visu_Ret_Arr[3] := FALSE;
   S702_HOOK_PIN.Visu_Ret_Arr[4] := FALSE;
   S702_HOOK_PIN.Visu_Ret_Arr[5] := FALSE;
   S702_HOOK_PIN.Visu_Ret_Arr[6] := FALSE;
   S702_HOOK_PIN.Visu_Ret_Arr[7] := FALSE;
   S702_HOOK_PIN.Visu_Ret_Arr[8] := FALSE;
   S702_HOOK_PIN.Visu_Ret_Arr[9] := FALSE;
   S702_HOOK_PIN.Visu_Ret_Arr[10] := FALSE;
   S702_HOOK_PIN.Visu_Ret_Arr[11] := FALSE;
   S702_HOOK_PIN.Visu_Ret_Arr[12] := FALSE;
   S702_HOOK_PIN.Visu_Ret_Arr[13] := FALSE;
   S702_HOOK_PIN.Visu_Ret_Arr[14] := FALSE;
   S702_HOOK_PIN.Visu_Ret_Arr[15] := FALSE;
   S702_HOOK_PIN.BLK_Move_Ret := 0;
   S702_HOOK_PIN.Enable := FALSE;
   S702_HOOK_PIN.Adv_End := FALSE;
   S702_HOOK_PIN.Ret_End := FALSE;
   S702_DAECHA_LOCK.Enable_Aux := FALSE;
   S702_DAECHA_LOCK.Adv_Amount := 0;
   S702_DAECHA_LOCK.Ret_Amount := 0;
   S702_DAECHA_LOCK.LS_Adv1 := FALSE;
   S702_DAECHA_LOCK.LS_Ret1 := FALSE;
   S702_DAECHA_LOCK.LS_Adv2 := FALSE;
   S702_DAECHA_LOCK.LS_Ret2 := FALSE;
   S702_DAECHA_LOCK.LS_Adv3 := FALSE;
   S702_DAECHA_LOCK.LS_Ret3 := FALSE;
   S702_DAECHA_LOCK.LS_Adv4 := FALSE;
   S702_DAECHA_LOCK.LS_Ret4 := FALSE;
   S702_DAECHA_LOCK.SOL_Adv := FALSE;
   S702_DAECHA_LOCK.SOL_Ret := FALSE;
   S702_DAECHA_LOCK.M_Ready := FALSE;
   S702_DAECHA_LOCK.T_CHK1 := T#0MS;
   S702_DAECHA_LOCK.T_CHK2 := T#0MS;
   S702_DAECHA_LOCK.PB_Lamp_CHK := FALSE;
   S702_DAECHA_LOCK.PB_Error_Rst := FALSE;
   S702_DAECHA_LOCK.M_FLICK := FALSE;
   S702_DAECHA_LOCK.M_Adv_Err := FALSE;
   S702_DAECHA_LOCK.M_Ret_Err := FALSE;
   S702_DAECHA_LOCK.LP_Adv := FALSE;
   S702_DAECHA_LOCK.LP_Ret := FALSE;
   S702_DAECHA_LOCK.Visu_Adv := W#16#0;
   S702_DAECHA_LOCK.Visu_Ret := W#16#0;
   S702_DAECHA_LOCK.Error_T1.IN := FALSE;
   S702_DAECHA_LOCK.Error_T1.PT := T#0MS;
   S702_DAECHA_LOCK.Error_T1.Q := FALSE;
   S702_DAECHA_LOCK.Error_T1.ET := T#0MS;
   S702_DAECHA_LOCK.Error_T1.STATE := B#16#0;
   S702_DAECHA_LOCK.Error_T1.STIME := T#0MS;
   S702_DAECHA_LOCK.Error_T1.ATIME := T#0MS;
   S702_DAECHA_LOCK.Error_T2.IN := FALSE;
   S702_DAECHA_LOCK.Error_T2.PT := T#0MS;
   S702_DAECHA_LOCK.Error_T2.Q := FALSE;
   S702_DAECHA_LOCK.Error_T2.ET := T#0MS;
   S702_DAECHA_LOCK.Error_T2.STATE := B#16#0;
   S702_DAECHA_LOCK.Error_T2.STIME := T#0MS;
   S702_DAECHA_LOCK.Error_T2.ATIME := T#0MS;
   S702_DAECHA_LOCK.CHK_Aux1 := FALSE;
   S702_DAECHA_LOCK.CHK_Aux2 := FALSE;
   S702_DAECHA_LOCK.Error_T1_DN := FALSE;
   S702_DAECHA_LOCK.Error_T2_DN := FALSE;
   S702_DAECHA_LOCK.Adv_Memo := FALSE;
   S702_DAECHA_LOCK.Visu_Adv_Arr[0] := FALSE;
   S702_DAECHA_LOCK.Visu_Adv_Arr[1] := FALSE;
   S702_DAECHA_LOCK.Visu_Adv_Arr[2] := FALSE;
   S702_DAECHA_LOCK.Visu_Adv_Arr[3] := FALSE;
   S702_DAECHA_LOCK.Visu_Adv_Arr[4] := FALSE;
   S702_DAECHA_LOCK.Visu_Adv_Arr[5] := FALSE;
   S702_DAECHA_LOCK.Visu_Adv_Arr[6] := FALSE;
   S702_DAECHA_LOCK.Visu_Adv_Arr[7] := FALSE;
   S702_DAECHA_LOCK.Visu_Adv_Arr[8] := FALSE;
   S702_DAECHA_LOCK.Visu_Adv_Arr[9] := FALSE;
   S702_DAECHA_LOCK.Visu_Adv_Arr[10] := FALSE;
   S702_DAECHA_LOCK.Visu_Adv_Arr[11] := FALSE;
   S702_DAECHA_LOCK.Visu_Adv_Arr[12] := FALSE;
   S702_DAECHA_LOCK.Visu_Adv_Arr[13] := FALSE;
   S702_DAECHA_LOCK.Visu_Adv_Arr[14] := FALSE;
   S702_DAECHA_LOCK.Visu_Adv_Arr[15] := FALSE;
   S702_DAECHA_LOCK.Visu_Ret_Arr[0] := FALSE;
   S702_DAECHA_LOCK.Visu_Ret_Arr[1] := FALSE;
   S702_DAECHA_LOCK.Visu_Ret_Arr[2] := FALSE;
   S702_DAECHA_LOCK.Visu_Ret_Arr[3] := FALSE;
   S702_DAECHA_LOCK.Visu_Ret_Arr[4] := FALSE;
   S702_DAECHA_LOCK.Visu_Ret_Arr[5] := FALSE;
   S702_DAECHA_LOCK.Visu_Ret_Arr[6] := FALSE;
   S702_DAECHA_LOCK.Visu_Ret_Arr[7] := FALSE;
   S702_DAECHA_LOCK.Visu_Ret_Arr[8] := FALSE;
   S702_DAECHA_LOCK.Visu_Ret_Arr[9] := FALSE;
   S702_DAECHA_LOCK.Visu_Ret_Arr[10] := FALSE;
   S702_DAECHA_LOCK.Visu_Ret_Arr[11] := FALSE;
   S702_DAECHA_LOCK.Visu_Ret_Arr[12] := FALSE;
   S702_DAECHA_LOCK.Visu_Ret_Arr[13] := FALSE;
   S702_DAECHA_LOCK.Visu_Ret_Arr[14] := FALSE;
   S702_DAECHA_LOCK.Visu_Ret_Arr[15] := FALSE;
   S702_DAECHA_LOCK.BLK_Move_Ret := 0;
   S702_DAECHA_LOCK.Enable := FALSE;
   S702_DAECHA_LOCK.Adv_End := FALSE;
   S702_DAECHA_LOCK.Ret_End := FALSE;
   S702_DAECHA_LOCK_UP_DN.Enable_Aux := FALSE;
   S702_DAECHA_LOCK_UP_DN.Adv_Amount := 0;
   S702_DAECHA_LOCK_UP_DN.Ret_Amount := 0;
   S702_DAECHA_LOCK_UP_DN.LS_Adv1 := FALSE;
   S702_DAECHA_LOCK_UP_DN.LS_Ret1 := FALSE;
   S702_DAECHA_LOCK_UP_DN.LS_Adv2 := FALSE;
   S702_DAECHA_LOCK_UP_DN.LS_Ret2 := FALSE;
   S702_DAECHA_LOCK_UP_DN.LS_Adv3 := FALSE;
   S702_DAECHA_LOCK_UP_DN.LS_Ret3 := FALSE;
   S702_DAECHA_LOCK_UP_DN.LS_Adv4 := FALSE;
   S702_DAECHA_LOCK_UP_DN.LS_Ret4 := FALSE;
   S702_DAECHA_LOCK_UP_DN.SOL_Adv := FALSE;
   S702_DAECHA_LOCK_UP_DN.SOL_Ret := FALSE;
   S702_DAECHA_LOCK_UP_DN.M_Ready := FALSE;
   S702_DAECHA_LOCK_UP_DN.T_CHK1 := T#0MS;
   S702_DAECHA_LOCK_UP_DN.T_CHK2 := T#0MS;
   S702_DAECHA_LOCK_UP_DN.PB_Lamp_CHK := FALSE;
   S702_DAECHA_LOCK_UP_DN.PB_Error_Rst := FALSE;
   S702_DAECHA_LOCK_UP_DN.M_FLICK := FALSE;
   S702_DAECHA_LOCK_UP_DN.M_Adv_Err := FALSE;
   S702_DAECHA_LOCK_UP_DN.M_Ret_Err := FALSE;
   S702_DAECHA_LOCK_UP_DN.LP_Adv := FALSE;
   S702_DAECHA_LOCK_UP_DN.LP_Ret := FALSE;
   S702_DAECHA_LOCK_UP_DN.Visu_Adv := W#16#0;
   S702_DAECHA_LOCK_UP_DN.Visu_Ret := W#16#0;
   S702_DAECHA_LOCK_UP_DN.Error_T1.IN := FALSE;
   S702_DAECHA_LOCK_UP_DN.Error_T1.PT := T#0MS;
   S702_DAECHA_LOCK_UP_DN.Error_T1.Q := FALSE;
   S702_DAECHA_LOCK_UP_DN.Error_T1.ET := T#0MS;
   S702_DAECHA_LOCK_UP_DN.Error_T1.STATE := B#16#0;
   S702_DAECHA_LOCK_UP_DN.Error_T1.STIME := T#0MS;
   S702_DAECHA_LOCK_UP_DN.Error_T1.ATIME := T#0MS;
   S702_DAECHA_LOCK_UP_DN.Error_T2.IN := FALSE;
   S702_DAECHA_LOCK_UP_DN.Error_T2.PT := T#0MS;
   S702_DAECHA_LOCK_UP_DN.Error_T2.Q := FALSE;
   S702_DAECHA_LOCK_UP_DN.Error_T2.ET := T#0MS;
   S702_DAECHA_LOCK_UP_DN.Error_T2.STATE := B#16#0;
   S702_DAECHA_LOCK_UP_DN.Error_T2.STIME := T#0MS;
   S702_DAECHA_LOCK_UP_DN.Error_T2.ATIME := T#0MS;
   S702_DAECHA_LOCK_UP_DN.CHK_Aux1 := FALSE;
   S702_DAECHA_LOCK_UP_DN.CHK_Aux2 := FALSE;
   S702_DAECHA_LOCK_UP_DN.Error_T1_DN := FALSE;
   S702_DAECHA_LOCK_UP_DN.Error_T2_DN := FALSE;
   S702_DAECHA_LOCK_UP_DN.Adv_Memo := FALSE;
   S702_DAECHA_LOCK_UP_DN.Visu_Adv_Arr[0] := FALSE;
   S702_DAECHA_LOCK_UP_DN.Visu_Adv_Arr[1] := FALSE;
   S702_DAECHA_LOCK_UP_DN.Visu_Adv_Arr[2] := FALSE;
   S702_DAECHA_LOCK_UP_DN.Visu_Adv_Arr[3] := FALSE;
   S702_DAECHA_LOCK_UP_DN.Visu_Adv_Arr[4] := FALSE;
   S702_DAECHA_LOCK_UP_DN.Visu_Adv_Arr[5] := FALSE;
   S702_DAECHA_LOCK_UP_DN.Visu_Adv_Arr[6] := FALSE;
   S702_DAECHA_LOCK_UP_DN.Visu_Adv_Arr[7] := FALSE;
   S702_DAECHA_LOCK_UP_DN.Visu_Adv_Arr[8] := FALSE;
   S702_DAECHA_LOCK_UP_DN.Visu_Adv_Arr[9] := FALSE;
   S702_DAECHA_LOCK_UP_DN.Visu_Adv_Arr[10] := FALSE;
   S702_DAECHA_LOCK_UP_DN.Visu_Adv_Arr[11] := FALSE;
   S702_DAECHA_LOCK_UP_DN.Visu_Adv_Arr[12] := FALSE;
   S702_DAECHA_LOCK_UP_DN.Visu_Adv_Arr[13] := FALSE;
   S702_DAECHA_LOCK_UP_DN.Visu_Adv_Arr[14] := FALSE;
   S702_DAECHA_LOCK_UP_DN.Visu_Adv_Arr[15] := FALSE;
   S702_DAECHA_LOCK_UP_DN.Visu_Ret_Arr[0] := FALSE;
   S702_DAECHA_LOCK_UP_DN.Visu_Ret_Arr[1] := FALSE;
   S702_DAECHA_LOCK_UP_DN.Visu_Ret_Arr[2] := FALSE;
   S702_DAECHA_LOCK_UP_DN.Visu_Ret_Arr[3] := FALSE;
   S702_DAECHA_LOCK_UP_DN.Visu_Ret_Arr[4] := FALSE;
   S702_DAECHA_LOCK_UP_DN.Visu_Ret_Arr[5] := FALSE;
   S702_DAECHA_LOCK_UP_DN.Visu_Ret_Arr[6] := FALSE;
   S702_DAECHA_LOCK_UP_DN.Visu_Ret_Arr[7] := FALSE;
   S702_DAECHA_LOCK_UP_DN.Visu_Ret_Arr[8] := FALSE;
   S702_DAECHA_LOCK_UP_DN.Visu_Ret_Arr[9] := FALSE;
   S702_DAECHA_LOCK_UP_DN.Visu_Ret_Arr[10] := FALSE;
   S702_DAECHA_LOCK_UP_DN.Visu_Ret_Arr[11] := FALSE;
   S702_DAECHA_LOCK_UP_DN.Visu_Ret_Arr[12] := FALSE;
   S702_DAECHA_LOCK_UP_DN.Visu_Ret_Arr[13] := FALSE;
   S702_DAECHA_LOCK_UP_DN.Visu_Ret_Arr[14] := FALSE;
   S702_DAECHA_LOCK_UP_DN.Visu_Ret_Arr[15] := FALSE;
   S702_DAECHA_LOCK_UP_DN.BLK_Move_Ret := 0;
   S702_DAECHA_LOCK_UP_DN.Enable := FALSE;
   S702_DAECHA_LOCK_UP_DN.Adv_End := FALSE;
   S702_DAECHA_LOCK_UP_DN.Ret_End := FALSE;
   S702_ELE.Enable_Aux := FALSE;
   S702_ELE.Adv_Amount := 0;
   S702_ELE.Ret_Amount := 0;
   S702_ELE.LS_Adv1 := FALSE;
   S702_ELE.LS_Ret1 := FALSE;
   S702_ELE.LS_Adv2 := FALSE;
   S702_ELE.LS_Ret2 := FALSE;
   S702_ELE.LS_Adv3 := FALSE;
   S702_ELE.LS_Ret3 := FALSE;
   S702_ELE.LS_Adv4 := FALSE;
   S702_ELE.LS_Ret4 := FALSE;
   S702_ELE.SOL_Adv := FALSE;
   S702_ELE.SOL_Ret := FALSE;
   S702_ELE.M_Ready := FALSE;
   S702_ELE.T_CHK1 := T#0MS;
   S702_ELE.T_CHK2 := T#0MS;
   S702_ELE.PB_Lamp_CHK := FALSE;
   S702_ELE.PB_Error_Rst := FALSE;
   S702_ELE.M_FLICK := FALSE;
   S702_ELE.M_Adv_Err := FALSE;
   S702_ELE.M_Ret_Err := FALSE;
   S702_ELE.LP_Adv := FALSE;
   S702_ELE.LP_Ret := FALSE;
   S702_ELE.Visu_Adv := W#16#0;
   S702_ELE.Visu_Ret := W#16#0;
   S702_ELE.Error_T1.IN := FALSE;
   S702_ELE.Error_T1.PT := T#0MS;
   S702_ELE.Error_T1.Q := FALSE;
   S702_ELE.Error_T1.ET := T#0MS;
   S702_ELE.Error_T1.STATE := B#16#0;
   S702_ELE.Error_T1.STIME := T#0MS;
   S702_ELE.Error_T1.ATIME := T#0MS;
   S702_ELE.Error_T2.IN := FALSE;
   S702_ELE.Error_T2.PT := T#0MS;
   S702_ELE.Error_T2.Q := FALSE;
   S702_ELE.Error_T2.ET := T#0MS;
   S702_ELE.Error_T2.STATE := B#16#0;
   S702_ELE.Error_T2.STIME := T#0MS;
   S702_ELE.Error_T2.ATIME := T#0MS;
   S702_ELE.CHK_Aux1 := FALSE;
   S702_ELE.CHK_Aux2 := FALSE;
   S702_ELE.Error_T1_DN := FALSE;
   S702_ELE.Error_T2_DN := FALSE;
   S702_ELE.Adv_Memo := FALSE;
   S702_ELE.Visu_Adv_Arr[0] := FALSE;
   S702_ELE.Visu_Adv_Arr[1] := FALSE;
   S702_ELE.Visu_Adv_Arr[2] := FALSE;
   S702_ELE.Visu_Adv_Arr[3] := FALSE;
   S702_ELE.Visu_Adv_Arr[4] := FALSE;
   S702_ELE.Visu_Adv_Arr[5] := FALSE;
   S702_ELE.Visu_Adv_Arr[6] := FALSE;
   S702_ELE.Visu_Adv_Arr[7] := FALSE;
   S702_ELE.Visu_Adv_Arr[8] := FALSE;
   S702_ELE.Visu_Adv_Arr[9] := FALSE;
   S702_ELE.Visu_Adv_Arr[10] := FALSE;
   S702_ELE.Visu_Adv_Arr[11] := FALSE;
   S702_ELE.Visu_Adv_Arr[12] := FALSE;
   S702_ELE.Visu_Adv_Arr[13] := FALSE;
   S702_ELE.Visu_Adv_Arr[14] := FALSE;
   S702_ELE.Visu_Adv_Arr[15] := FALSE;
   S702_ELE.Visu_Ret_Arr[0] := FALSE;
   S702_ELE.Visu_Ret_Arr[1] := FALSE;
   S702_ELE.Visu_Ret_Arr[2] := FALSE;
   S702_ELE.Visu_Ret_Arr[3] := FALSE;
   S702_ELE.Visu_Ret_Arr[4] := FALSE;
   S702_ELE.Visu_Ret_Arr[5] := FALSE;
   S702_ELE.Visu_Ret_Arr[6] := FALSE;
   S702_ELE.Visu_Ret_Arr[7] := FALSE;
   S702_ELE.Visu_Ret_Arr[8] := FALSE;
   S702_ELE.Visu_Ret_Arr[9] := FALSE;
   S702_ELE.Visu_Ret_Arr[10] := FALSE;
   S702_ELE.Visu_Ret_Arr[11] := FALSE;
   S702_ELE.Visu_Ret_Arr[12] := FALSE;
   S702_ELE.Visu_Ret_Arr[13] := FALSE;
   S702_ELE.Visu_Ret_Arr[14] := FALSE;
   S702_ELE.Visu_Ret_Arr[15] := FALSE;
   S702_ELE.BLK_Move_Ret := 0;
   S702_ELE.Enable := FALSE;
   S702_ELE.Adv_End := FALSE;
   S702_ELE.Ret_End := FALSE;
   S702_AIR_ELE.Enable_Aux := FALSE;
   S702_AIR_ELE.Adv_Amount := 0;
   S702_AIR_ELE.Ret_Amount := 0;
   S702_AIR_ELE.LS_Adv1 := FALSE;
   S702_AIR_ELE.LS_Ret1 := FALSE;
   S702_AIR_ELE.LS_Adv2 := FALSE;
   S702_AIR_ELE.LS_Ret2 := FALSE;
   S702_AIR_ELE.LS_Adv3 := FALSE;
   S702_AIR_ELE.LS_Ret3 := FALSE;
   S702_AIR_ELE.LS_Adv4 := FALSE;
   S702_AIR_ELE.LS_Ret4 := FALSE;
   S702_AIR_ELE.SOL_Adv := FALSE;
   S702_AIR_ELE.SOL_Ret := FALSE;
   S702_AIR_ELE.M_Ready := FALSE;
   S702_AIR_ELE.T_CHK1 := T#0MS;
   S702_AIR_ELE.T_CHK2 := T#0MS;
   S702_AIR_ELE.PB_Lamp_CHK := FALSE;
   S702_AIR_ELE.PB_Error_Rst := FALSE;
   S702_AIR_ELE.M_FLICK := FALSE;
   S702_AIR_ELE.M_Adv_Err := FALSE;
   S702_AIR_ELE.M_Ret_Err := FALSE;
   S702_AIR_ELE.LP_Adv := FALSE;
   S702_AIR_ELE.LP_Ret := FALSE;
   S702_AIR_ELE.Visu_Adv := W#16#0;
   S702_AIR_ELE.Visu_Ret := W#16#0;
   S702_AIR_ELE.Error_T1.IN := FALSE;
   S702_AIR_ELE.Error_T1.PT := T#0MS;
   S702_AIR_ELE.Error_T1.Q := FALSE;
   S702_AIR_ELE.Error_T1.ET := T#0MS;
   S702_AIR_ELE.Error_T1.STATE := B#16#0;
   S702_AIR_ELE.Error_T1.STIME := T#0MS;
   S702_AIR_ELE.Error_T1.ATIME := T#0MS;
   S702_AIR_ELE.Error_T2.IN := FALSE;
   S702_AIR_ELE.Error_T2.PT := T#0MS;
   S702_AIR_ELE.Error_T2.Q := FALSE;
   S702_AIR_ELE.Error_T2.ET := T#0MS;
   S702_AIR_ELE.Error_T2.STATE := B#16#0;
   S702_AIR_ELE.Error_T2.STIME := T#0MS;
   S702_AIR_ELE.Error_T2.ATIME := T#0MS;
   S702_AIR_ELE.CHK_Aux1 := FALSE;
   S702_AIR_ELE.CHK_Aux2 := FALSE;
   S702_AIR_ELE.Error_T1_DN := FALSE;
   S702_AIR_ELE.Error_T2_DN := FALSE;
   S702_AIR_ELE.Adv_Memo := FALSE;
   S702_AIR_ELE.Visu_Adv_Arr[0] := FALSE;
   S702_AIR_ELE.Visu_Adv_Arr[1] := FALSE;
   S702_AIR_ELE.Visu_Adv_Arr[2] := FALSE;
   S702_AIR_ELE.Visu_Adv_Arr[3] := FALSE;
   S702_AIR_ELE.Visu_Adv_Arr[4] := FALSE;
   S702_AIR_ELE.Visu_Adv_Arr[5] := FALSE;
   S702_AIR_ELE.Visu_Adv_Arr[6] := FALSE;
   S702_AIR_ELE.Visu_Adv_Arr[7] := FALSE;
   S702_AIR_ELE.Visu_Adv_Arr[8] := FALSE;
   S702_AIR_ELE.Visu_Adv_Arr[9] := FALSE;
   S702_AIR_ELE.Visu_Adv_Arr[10] := FALSE;
   S702_AIR_ELE.Visu_Adv_Arr[11] := FALSE;
   S702_AIR_ELE.Visu_Adv_Arr[12] := FALSE;
   S702_AIR_ELE.Visu_Adv_Arr[13] := FALSE;
   S702_AIR_ELE.Visu_Adv_Arr[14] := FALSE;
   S702_AIR_ELE.Visu_Adv_Arr[15] := FALSE;
   S702_AIR_ELE.Visu_Ret_Arr[0] := FALSE;
   S702_AIR_ELE.Visu_Ret_Arr[1] := FALSE;
   S702_AIR_ELE.Visu_Ret_Arr[2] := FALSE;
   S702_AIR_ELE.Visu_Ret_Arr[3] := FALSE;
   S702_AIR_ELE.Visu_Ret_Arr[4] := FALSE;
   S702_AIR_ELE.Visu_Ret_Arr[5] := FALSE;
   S702_AIR_ELE.Visu_Ret_Arr[6] := FALSE;
   S702_AIR_ELE.Visu_Ret_Arr[7] := FALSE;
   S702_AIR_ELE.Visu_Ret_Arr[8] := FALSE;
   S702_AIR_ELE.Visu_Ret_Arr[9] := FALSE;
   S702_AIR_ELE.Visu_Ret_Arr[10] := FALSE;
   S702_AIR_ELE.Visu_Ret_Arr[11] := FALSE;
   S702_AIR_ELE.Visu_Ret_Arr[12] := FALSE;
   S702_AIR_ELE.Visu_Ret_Arr[13] := FALSE;
   S702_AIR_ELE.Visu_Ret_Arr[14] := FALSE;
   S702_AIR_ELE.Visu_Ret_Arr[15] := FALSE;
   S702_AIR_ELE.BLK_Move_Ret := 0;
   S702_AIR_ELE.Enable := FALSE;
   S702_AIR_ELE.Adv_End := FALSE;
   S702_AIR_ELE.Ret_End := FALSE;
   S702_EJECT.Enable_Aux := FALSE;
   S702_EJECT.Adv_Amount := 0;
   S702_EJECT.Ret_Amount := 0;
   S702_EJECT.LS_Adv1 := FALSE;
   S702_EJECT.LS_Ret1 := FALSE;
   S702_EJECT.LS_Adv2 := FALSE;
   S702_EJECT.LS_Ret2 := FALSE;
   S702_EJECT.LS_Adv3 := FALSE;
   S702_EJECT.LS_Ret3 := FALSE;
   S702_EJECT.LS_Adv4 := FALSE;
   S702_EJECT.LS_Ret4 := FALSE;
   S702_EJECT.SOL_Adv := FALSE;
   S702_EJECT.SOL_Ret := FALSE;
   S702_EJECT.M_Ready := FALSE;
   S702_EJECT.T_CHK1 := T#0MS;
   S702_EJECT.T_CHK2 := T#0MS;
   S702_EJECT.PB_Lamp_CHK := FALSE;
   S702_EJECT.PB_Error_Rst := FALSE;
   S702_EJECT.M_FLICK := FALSE;
   S702_EJECT.M_Adv_Err := FALSE;
   S702_EJECT.M_Ret_Err := FALSE;
   S702_EJECT.LP_Adv := FALSE;
   S702_EJECT.LP_Ret := FALSE;
   S702_EJECT.Visu_Adv := W#16#0;
   S702_EJECT.Visu_Ret := W#16#0;
   S702_EJECT.Error_T1.IN := FALSE;
   S702_EJECT.Error_T1.PT := T#0MS;
   S702_EJECT.Error_T1.Q := FALSE;
   S702_EJECT.Error_T1.ET := T#0MS;
   S702_EJECT.Error_T1.STATE := B#16#0;
   S702_EJECT.Error_T1.STIME := T#0MS;
   S702_EJECT.Error_T1.ATIME := T#0MS;
   S702_EJECT.Error_T2.IN := FALSE;
   S702_EJECT.Error_T2.PT := T#0MS;
   S702_EJECT.Error_T2.Q := FALSE;
   S702_EJECT.Error_T2.ET := T#0MS;
   S702_EJECT.Error_T2.STATE := B#16#0;
   S702_EJECT.Error_T2.STIME := T#0MS;
   S702_EJECT.Error_T2.ATIME := T#0MS;
   S702_EJECT.CHK_Aux1 := FALSE;
   S702_EJECT.CHK_Aux2 := FALSE;
   S702_EJECT.Error_T1_DN := FALSE;
   S702_EJECT.Error_T2_DN := FALSE;
   S702_EJECT.Adv_Memo := FALSE;
   S702_EJECT.Visu_Adv_Arr[0] := FALSE;
   S702_EJECT.Visu_Adv_Arr[1] := FALSE;
   S702_EJECT.Visu_Adv_Arr[2] := FALSE;
   S702_EJECT.Visu_Adv_Arr[3] := FALSE;
   S702_EJECT.Visu_Adv_Arr[4] := FALSE;
   S702_EJECT.Visu_Adv_Arr[5] := FALSE;
   S702_EJECT.Visu_Adv_Arr[6] := FALSE;
   S702_EJECT.Visu_Adv_Arr[7] := FALSE;
   S702_EJECT.Visu_Adv_Arr[8] := FALSE;
   S702_EJECT.Visu_Adv_Arr[9] := FALSE;
   S702_EJECT.Visu_Adv_Arr[10] := FALSE;
   S702_EJECT.Visu_Adv_Arr[11] := FALSE;
   S702_EJECT.Visu_Adv_Arr[12] := FALSE;
   S702_EJECT.Visu_Adv_Arr[13] := FALSE;
   S702_EJECT.Visu_Adv_Arr[14] := FALSE;
   S702_EJECT.Visu_Adv_Arr[15] := FALSE;
   S702_EJECT.Visu_Ret_Arr[0] := FALSE;
   S702_EJECT.Visu_Ret_Arr[1] := FALSE;
   S702_EJECT.Visu_Ret_Arr[2] := FALSE;
   S702_EJECT.Visu_Ret_Arr[3] := FALSE;
   S702_EJECT.Visu_Ret_Arr[4] := FALSE;
   S702_EJECT.Visu_Ret_Arr[5] := FALSE;
   S702_EJECT.Visu_Ret_Arr[6] := FALSE;
   S702_EJECT.Visu_Ret_Arr[7] := FALSE;
   S702_EJECT.Visu_Ret_Arr[8] := FALSE;
   S702_EJECT.Visu_Ret_Arr[9] := FALSE;
   S702_EJECT.Visu_Ret_Arr[10] := FALSE;
   S702_EJECT.Visu_Ret_Arr[11] := FALSE;
   S702_EJECT.Visu_Ret_Arr[12] := FALSE;
   S702_EJECT.Visu_Ret_Arr[13] := FALSE;
   S702_EJECT.Visu_Ret_Arr[14] := FALSE;
   S702_EJECT.Visu_Ret_Arr[15] := FALSE;
   S702_EJECT.BLK_Move_Ret := 0;
   S702_EJECT.Enable := FALSE;
   S702_EJECT.Adv_End := FALSE;
   S702_EJECT.Ret_End := FALSE;
   S702_DAECHA_STOPPER.Enable_Aux := FALSE;
   S702_DAECHA_STOPPER.Adv_Amount := 0;
   S702_DAECHA_STOPPER.Ret_Amount := 0;
   S702_DAECHA_STOPPER.LS_Adv1 := FALSE;
   S702_DAECHA_STOPPER.LS_Ret1 := FALSE;
   S702_DAECHA_STOPPER.LS_Adv2 := FALSE;
   S702_DAECHA_STOPPER.LS_Ret2 := FALSE;
   S702_DAECHA_STOPPER.LS_Adv3 := FALSE;
   S702_DAECHA_STOPPER.LS_Ret3 := FALSE;
   S702_DAECHA_STOPPER.LS_Adv4 := FALSE;
   S702_DAECHA_STOPPER.LS_Ret4 := FALSE;
   S702_DAECHA_STOPPER.SOL_Adv := FALSE;
   S702_DAECHA_STOPPER.SOL_Ret := FALSE;
   S702_DAECHA_STOPPER.M_Ready := FALSE;
   S702_DAECHA_STOPPER.T_CHK1 := T#0MS;
   S702_DAECHA_STOPPER.T_CHK2 := T#0MS;
   S702_DAECHA_STOPPER.PB_Lamp_CHK := FALSE;
   S702_DAECHA_STOPPER.PB_Error_Rst := FALSE;
   S702_DAECHA_STOPPER.M_FLICK := FALSE;
   S702_DAECHA_STOPPER.M_Adv_Err := FALSE;
   S702_DAECHA_STOPPER.M_Ret_Err := FALSE;
   S702_DAECHA_STOPPER.LP_Adv := FALSE;
   S702_DAECHA_STOPPER.LP_Ret := FALSE;
   S702_DAECHA_STOPPER.Visu_Adv := W#16#0;
   S702_DAECHA_STOPPER.Visu_Ret := W#16#0;
   S702_DAECHA_STOPPER.Error_T1.IN := FALSE;
   S702_DAECHA_STOPPER.Error_T1.PT := T#0MS;
   S702_DAECHA_STOPPER.Error_T1.Q := FALSE;
   S702_DAECHA_STOPPER.Error_T1.ET := T#0MS;
   S702_DAECHA_STOPPER.Error_T1.STATE := B#16#0;
   S702_DAECHA_STOPPER.Error_T1.STIME := T#0MS;
   S702_DAECHA_STOPPER.Error_T1.ATIME := T#0MS;
   S702_DAECHA_STOPPER.Error_T2.IN := FALSE;
   S702_DAECHA_STOPPER.Error_T2.PT := T#0MS;
   S702_DAECHA_STOPPER.Error_T2.Q := FALSE;
   S702_DAECHA_STOPPER.Error_T2.ET := T#0MS;
   S702_DAECHA_STOPPER.Error_T2.STATE := B#16#0;
   S702_DAECHA_STOPPER.Error_T2.STIME := T#0MS;
   S702_DAECHA_STOPPER.Error_T2.ATIME := T#0MS;
   S702_DAECHA_STOPPER.CHK_Aux1 := FALSE;
   S702_DAECHA_STOPPER.CHK_Aux2 := FALSE;
   S702_DAECHA_STOPPER.Error_T1_DN := FALSE;
   S702_DAECHA_STOPPER.Error_T2_DN := FALSE;
   S702_DAECHA_STOPPER.Adv_Memo := FALSE;
   S702_DAECHA_STOPPER.Visu_Adv_Arr[0] := FALSE;
   S702_DAECHA_STOPPER.Visu_Adv_Arr[1] := FALSE;
   S702_DAECHA_STOPPER.Visu_Adv_Arr[2] := FALSE;
   S702_DAECHA_STOPPER.Visu_Adv_Arr[3] := FALSE;
   S702_DAECHA_STOPPER.Visu_Adv_Arr[4] := FALSE;
   S702_DAECHA_STOPPER.Visu_Adv_Arr[5] := FALSE;
   S702_DAECHA_STOPPER.Visu_Adv_Arr[6] := FALSE;
   S702_DAECHA_STOPPER.Visu_Adv_Arr[7] := FALSE;
   S702_DAECHA_STOPPER.Visu_Adv_Arr[8] := FALSE;
   S702_DAECHA_STOPPER.Visu_Adv_Arr[9] := FALSE;
   S702_DAECHA_STOPPER.Visu_Adv_Arr[10] := FALSE;
   S702_DAECHA_STOPPER.Visu_Adv_Arr[11] := FALSE;
   S702_DAECHA_STOPPER.Visu_Adv_Arr[12] := FALSE;
   S702_DAECHA_STOPPER.Visu_Adv_Arr[13] := FALSE;
   S702_DAECHA_STOPPER.Visu_Adv_Arr[14] := FALSE;
   S702_DAECHA_STOPPER.Visu_Adv_Arr[15] := FALSE;
   S702_DAECHA_STOPPER.Visu_Ret_Arr[0] := FALSE;
   S702_DAECHA_STOPPER.Visu_Ret_Arr[1] := FALSE;
   S702_DAECHA_STOPPER.Visu_Ret_Arr[2] := FALSE;
   S702_DAECHA_STOPPER.Visu_Ret_Arr[3] := FALSE;
   S702_DAECHA_STOPPER.Visu_Ret_Arr[4] := FALSE;
   S702_DAECHA_STOPPER.Visu_Ret_Arr[5] := FALSE;
   S702_DAECHA_STOPPER.Visu_Ret_Arr[6] := FALSE;
   S702_DAECHA_STOPPER.Visu_Ret_Arr[7] := FALSE;
   S702_DAECHA_STOPPER.Visu_Ret_Arr[8] := FALSE;
   S702_DAECHA_STOPPER.Visu_Ret_Arr[9] := FALSE;
   S702_DAECHA_STOPPER.Visu_Ret_Arr[10] := FALSE;
   S702_DAECHA_STOPPER.Visu_Ret_Arr[11] := FALSE;
   S702_DAECHA_STOPPER.Visu_Ret_Arr[12] := FALSE;
   S702_DAECHA_STOPPER.Visu_Ret_Arr[13] := FALSE;
   S702_DAECHA_STOPPER.Visu_Ret_Arr[14] := FALSE;
   S702_DAECHA_STOPPER.Visu_Ret_Arr[15] := FALSE;
   S702_DAECHA_STOPPER.BLK_Move_Ret := 0;
   S702_DAECHA_STOPPER.Enable := FALSE;
   S702_DAECHA_STOPPER.Adv_End := FALSE;
   S702_DAECHA_STOPPER.Ret_End := FALSE;
   S702_DAECHA_CLAMP.Enable_Aux := FALSE;
   S702_DAECHA_CLAMP.Adv_Amount := 0;
   S702_DAECHA_CLAMP.Ret_Amount := 0;
   S702_DAECHA_CLAMP.LS_Adv1 := FALSE;
   S702_DAECHA_CLAMP.LS_Ret1 := FALSE;
   S702_DAECHA_CLAMP.LS_Adv2 := FALSE;
   S702_DAECHA_CLAMP.LS_Ret2 := FALSE;
   S702_DAECHA_CLAMP.LS_Adv3 := FALSE;
   S702_DAECHA_CLAMP.LS_Ret3 := FALSE;
   S702_DAECHA_CLAMP.LS_Adv4 := FALSE;
   S702_DAECHA_CLAMP.LS_Ret4 := FALSE;
   S702_DAECHA_CLAMP.SOL_Adv := FALSE;
   S702_DAECHA_CLAMP.SOL_Ret := FALSE;
   S702_DAECHA_CLAMP.M_Ready := FALSE;
   S702_DAECHA_CLAMP.T_CHK1 := T#0MS;
   S702_DAECHA_CLAMP.T_CHK2 := T#0MS;
   S702_DAECHA_CLAMP.PB_Lamp_CHK := FALSE;
   S702_DAECHA_CLAMP.PB_Error_Rst := FALSE;
   S702_DAECHA_CLAMP.M_FLICK := FALSE;
   S702_DAECHA_CLAMP.M_Adv_Err := FALSE;
   S702_DAECHA_CLAMP.M_Ret_Err := FALSE;
   S702_DAECHA_CLAMP.LP_Adv := FALSE;
   S702_DAECHA_CLAMP.LP_Ret := FALSE;
   S702_DAECHA_CLAMP.Visu_Adv := W#16#0;
   S702_DAECHA_CLAMP.Visu_Ret := W#16#0;
   S702_DAECHA_CLAMP.Error_T1.IN := FALSE;
   S702_DAECHA_CLAMP.Error_T1.PT := T#0MS;
   S702_DAECHA_CLAMP.Error_T1.Q := FALSE;
   S702_DAECHA_CLAMP.Error_T1.ET := T#0MS;
   S702_DAECHA_CLAMP.Error_T1.STATE := B#16#0;
   S702_DAECHA_CLAMP.Error_T1.STIME := T#0MS;
   S702_DAECHA_CLAMP.Error_T1.ATIME := T#0MS;
   S702_DAECHA_CLAMP.Error_T2.IN := FALSE;
   S702_DAECHA_CLAMP.Error_T2.PT := T#0MS;
   S702_DAECHA_CLAMP.Error_T2.Q := FALSE;
   S702_DAECHA_CLAMP.Error_T2.ET := T#0MS;
   S702_DAECHA_CLAMP.Error_T2.STATE := B#16#0;
   S702_DAECHA_CLAMP.Error_T2.STIME := T#0MS;
   S702_DAECHA_CLAMP.Error_T2.ATIME := T#0MS;
   S702_DAECHA_CLAMP.CHK_Aux1 := FALSE;
   S702_DAECHA_CLAMP.CHK_Aux2 := FALSE;
   S702_DAECHA_CLAMP.Error_T1_DN := FALSE;
   S702_DAECHA_CLAMP.Error_T2_DN := FALSE;
   S702_DAECHA_CLAMP.Adv_Memo := FALSE;
   S702_DAECHA_CLAMP.Visu_Adv_Arr[0] := FALSE;
   S702_DAECHA_CLAMP.Visu_Adv_Arr[1] := FALSE;
   S702_DAECHA_CLAMP.Visu_Adv_Arr[2] := FALSE;
   S702_DAECHA_CLAMP.Visu_Adv_Arr[3] := FALSE;
   S702_DAECHA_CLAMP.Visu_Adv_Arr[4] := FALSE;
   S702_DAECHA_CLAMP.Visu_Adv_Arr[5] := FALSE;
   S702_DAECHA_CLAMP.Visu_Adv_Arr[6] := FALSE;
   S702_DAECHA_CLAMP.Visu_Adv_Arr[7] := FALSE;
   S702_DAECHA_CLAMP.Visu_Adv_Arr[8] := FALSE;
   S702_DAECHA_CLAMP.Visu_Adv_Arr[9] := FALSE;
   S702_DAECHA_CLAMP.Visu_Adv_Arr[10] := FALSE;
   S702_DAECHA_CLAMP.Visu_Adv_Arr[11] := FALSE;
   S702_DAECHA_CLAMP.Visu_Adv_Arr[12] := FALSE;
   S702_DAECHA_CLAMP.Visu_Adv_Arr[13] := FALSE;
   S702_DAECHA_CLAMP.Visu_Adv_Arr[14] := FALSE;
   S702_DAECHA_CLAMP.Visu_Adv_Arr[15] := FALSE;
   S702_DAECHA_CLAMP.Visu_Ret_Arr[0] := FALSE;
   S702_DAECHA_CLAMP.Visu_Ret_Arr[1] := FALSE;
   S702_DAECHA_CLAMP.Visu_Ret_Arr[2] := FALSE;
   S702_DAECHA_CLAMP.Visu_Ret_Arr[3] := FALSE;
   S702_DAECHA_CLAMP.Visu_Ret_Arr[4] := FALSE;
   S702_DAECHA_CLAMP.Visu_Ret_Arr[5] := FALSE;
   S702_DAECHA_CLAMP.Visu_Ret_Arr[6] := FALSE;
   S702_DAECHA_CLAMP.Visu_Ret_Arr[7] := FALSE;
   S702_DAECHA_CLAMP.Visu_Ret_Arr[8] := FALSE;
   S702_DAECHA_CLAMP.Visu_Ret_Arr[9] := FALSE;
   S702_DAECHA_CLAMP.Visu_Ret_Arr[10] := FALSE;
   S702_DAECHA_CLAMP.Visu_Ret_Arr[11] := FALSE;
   S702_DAECHA_CLAMP.Visu_Ret_Arr[12] := FALSE;
   S702_DAECHA_CLAMP.Visu_Ret_Arr[13] := FALSE;
   S702_DAECHA_CLAMP.Visu_Ret_Arr[14] := FALSE;
   S702_DAECHA_CLAMP.Visu_Ret_Arr[15] := FALSE;
   S702_DAECHA_CLAMP.BLK_Move_Ret := 0;
   S702_DAECHA_CLAMP.Enable := FALSE;
   S702_DAECHA_CLAMP.Adv_End := FALSE;
   S702_DAECHA_CLAMP.Ret_End := FALSE;
   S702_SHOCK_ABSORBER.Enable_Aux := FALSE;
   S702_SHOCK_ABSORBER.Adv_Amount := 0;
   S702_SHOCK_ABSORBER.Ret_Amount := 0;
   S702_SHOCK_ABSORBER.LS_Adv1 := FALSE;
   S702_SHOCK_ABSORBER.LS_Ret1 := FALSE;
   S702_SHOCK_ABSORBER.LS_Adv2 := FALSE;
   S702_SHOCK_ABSORBER.LS_Ret2 := FALSE;
   S702_SHOCK_ABSORBER.LS_Adv3 := FALSE;
   S702_SHOCK_ABSORBER.LS_Ret3 := FALSE;
   S702_SHOCK_ABSORBER.LS_Adv4 := FALSE;
   S702_SHOCK_ABSORBER.LS_Ret4 := FALSE;
   S702_SHOCK_ABSORBER.SOL_Adv := FALSE;
   S702_SHOCK_ABSORBER.SOL_Ret := FALSE;
   S702_SHOCK_ABSORBER.M_Ready := FALSE;
   S702_SHOCK_ABSORBER.T_CHK1 := T#0MS;
   S702_SHOCK_ABSORBER.T_CHK2 := T#0MS;
   S702_SHOCK_ABSORBER.PB_Lamp_CHK := FALSE;
   S702_SHOCK_ABSORBER.PB_Error_Rst := FALSE;
   S702_SHOCK_ABSORBER.M_FLICK := FALSE;
   S702_SHOCK_ABSORBER.M_Adv_Err := FALSE;
   S702_SHOCK_ABSORBER.M_Ret_Err := FALSE;
   S702_SHOCK_ABSORBER.LP_Adv := FALSE;
   S702_SHOCK_ABSORBER.LP_Ret := FALSE;
   S702_SHOCK_ABSORBER.Visu_Adv := W#16#0;
   S702_SHOCK_ABSORBER.Visu_Ret := W#16#0;
   S702_SHOCK_ABSORBER.Error_T1.IN := FALSE;
   S702_SHOCK_ABSORBER.Error_T1.PT := T#0MS;
   S702_SHOCK_ABSORBER.Error_T1.Q := FALSE;
   S702_SHOCK_ABSORBER.Error_T1.ET := T#0MS;
   S702_SHOCK_ABSORBER.Error_T1.STATE := B#16#0;
   S702_SHOCK_ABSORBER.Error_T1.STIME := T#0MS;
   S702_SHOCK_ABSORBER.Error_T1.ATIME := T#0MS;
   S702_SHOCK_ABSORBER.Error_T2.IN := FALSE;
   S702_SHOCK_ABSORBER.Error_T2.PT := T#0MS;
   S702_SHOCK_ABSORBER.Error_T2.Q := FALSE;
   S702_SHOCK_ABSORBER.Error_T2.ET := T#0MS;
   S702_SHOCK_ABSORBER.Error_T2.STATE := B#16#0;
   S702_SHOCK_ABSORBER.Error_T2.STIME := T#0MS;
   S702_SHOCK_ABSORBER.Error_T2.ATIME := T#0MS;
   S702_SHOCK_ABSORBER.CHK_Aux1 := FALSE;
   S702_SHOCK_ABSORBER.CHK_Aux2 := FALSE;
   S702_SHOCK_ABSORBER.Error_T1_DN := FALSE;
   S702_SHOCK_ABSORBER.Error_T2_DN := FALSE;
   S702_SHOCK_ABSORBER.Adv_Memo := FALSE;
   S702_SHOCK_ABSORBER.Visu_Adv_Arr[0] := FALSE;
   S702_SHOCK_ABSORBER.Visu_Adv_Arr[1] := FALSE;
   S702_SHOCK_ABSORBER.Visu_Adv_Arr[2] := FALSE;
   S702_SHOCK_ABSORBER.Visu_Adv_Arr[3] := FALSE;
   S702_SHOCK_ABSORBER.Visu_Adv_Arr[4] := FALSE;
   S702_SHOCK_ABSORBER.Visu_Adv_Arr[5] := FALSE;
   S702_SHOCK_ABSORBER.Visu_Adv_Arr[6] := FALSE;
   S702_SHOCK_ABSORBER.Visu_Adv_Arr[7] := FALSE;
   S702_SHOCK_ABSORBER.Visu_Adv_Arr[8] := FALSE;
   S702_SHOCK_ABSORBER.Visu_Adv_Arr[9] := FALSE;
   S702_SHOCK_ABSORBER.Visu_Adv_Arr[10] := FALSE;
   S702_SHOCK_ABSORBER.Visu_Adv_Arr[11] := FALSE;
   S702_SHOCK_ABSORBER.Visu_Adv_Arr[12] := FALSE;
   S702_SHOCK_ABSORBER.Visu_Adv_Arr[13] := FALSE;
   S702_SHOCK_ABSORBER.Visu_Adv_Arr[14] := FALSE;
   S702_SHOCK_ABSORBER.Visu_Adv_Arr[15] := FALSE;
   S702_SHOCK_ABSORBER.Visu_Ret_Arr[0] := FALSE;
   S702_SHOCK_ABSORBER.Visu_Ret_Arr[1] := FALSE;
   S702_SHOCK_ABSORBER.Visu_Ret_Arr[2] := FALSE;
   S702_SHOCK_ABSORBER.Visu_Ret_Arr[3] := FALSE;
   S702_SHOCK_ABSORBER.Visu_Ret_Arr[4] := FALSE;
   S702_SHOCK_ABSORBER.Visu_Ret_Arr[5] := FALSE;
   S702_SHOCK_ABSORBER.Visu_Ret_Arr[6] := FALSE;
   S702_SHOCK_ABSORBER.Visu_Ret_Arr[7] := FALSE;
   S702_SHOCK_ABSORBER.Visu_Ret_Arr[8] := FALSE;
   S702_SHOCK_ABSORBER.Visu_Ret_Arr[9] := FALSE;
   S702_SHOCK_ABSORBER.Visu_Ret_Arr[10] := FALSE;
   S702_SHOCK_ABSORBER.Visu_Ret_Arr[11] := FALSE;
   S702_SHOCK_ABSORBER.Visu_Ret_Arr[12] := FALSE;
   S702_SHOCK_ABSORBER.Visu_Ret_Arr[13] := FALSE;
   S702_SHOCK_ABSORBER.Visu_Ret_Arr[14] := FALSE;
   S702_SHOCK_ABSORBER.Visu_Ret_Arr[15] := FALSE;
   S702_SHOCK_ABSORBER.BLK_Move_Ret := 0;
   S702_SHOCK_ABSORBER.Enable := FALSE;
   S702_SHOCK_ABSORBER.Adv_End := FALSE;
   S702_SHOCK_ABSORBER.Ret_End := FALSE;
END_DATA_BLOCK

FUNCTION FC 121 : VOID
TITLE =
VERSION : 0.1

BEGIN
NETWORK
TITLE =
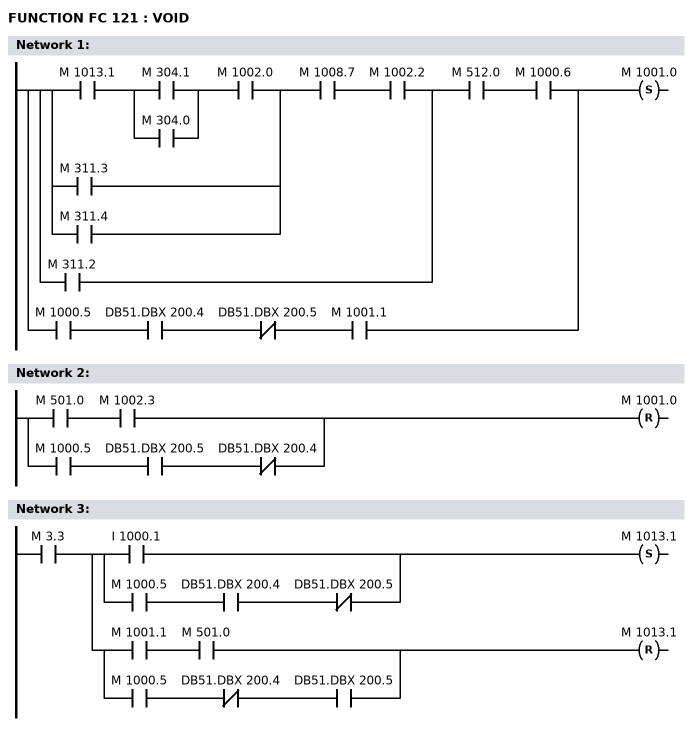

      A(    ;
      A(    ;
      A     M   1013.1;
      A(    ;
      O     M    304.1;
      O     M    304.0;
      )     ;
      A     M   1002.0;
      O     M    311.3;
      O     M    311.4;
      )     ;
      A     M   1008.7;
      A     M   1002.2;
      O     M    311.2;
      )     ;
      A     M    512.0;
      A     M   1000.6;
      O     ;
      A     M   1000.5;
      A     DB51.DBX  200.4;
      AN    DB51.DBX  200.5;
      A     M   1001.1;
      S     M   1001.0;
NETWORK
TITLE =

      A     M    501.0;
      A     M   1002.3;
      O     ;
      A     M   1000.5;
      A     DB51.DBX  200.5;
      AN    DB51.DBX  200.4;
      R     M   1001.0;
NETWORK
TITLE =

      A     M      3.3;
      =     L      0.0;
      A     L      0.0;
      A(    ;
      O     I   1000.1;
      O     ;
      A     M   1000.5;
      A     DB51.DBX  200.4;
      AN    DB51.DBX  200.5;
      )     ;
      S     M   1013.1;
      A     L      0.0;
      A(    ;
      A     M   1001.1;
      A     M    501.0;
      O     ;
      A     M   1000.5;
      AN    DB51.DBX  200.4;
      A     DB51.DBX  200.5;
      )     ;
      R     M   1013.1;
END_FUNCTION

FUNCTION_BLOCK FB 122
TITLE =
VERSION : 0.1

BEGIN
NETWORK
TITLE =
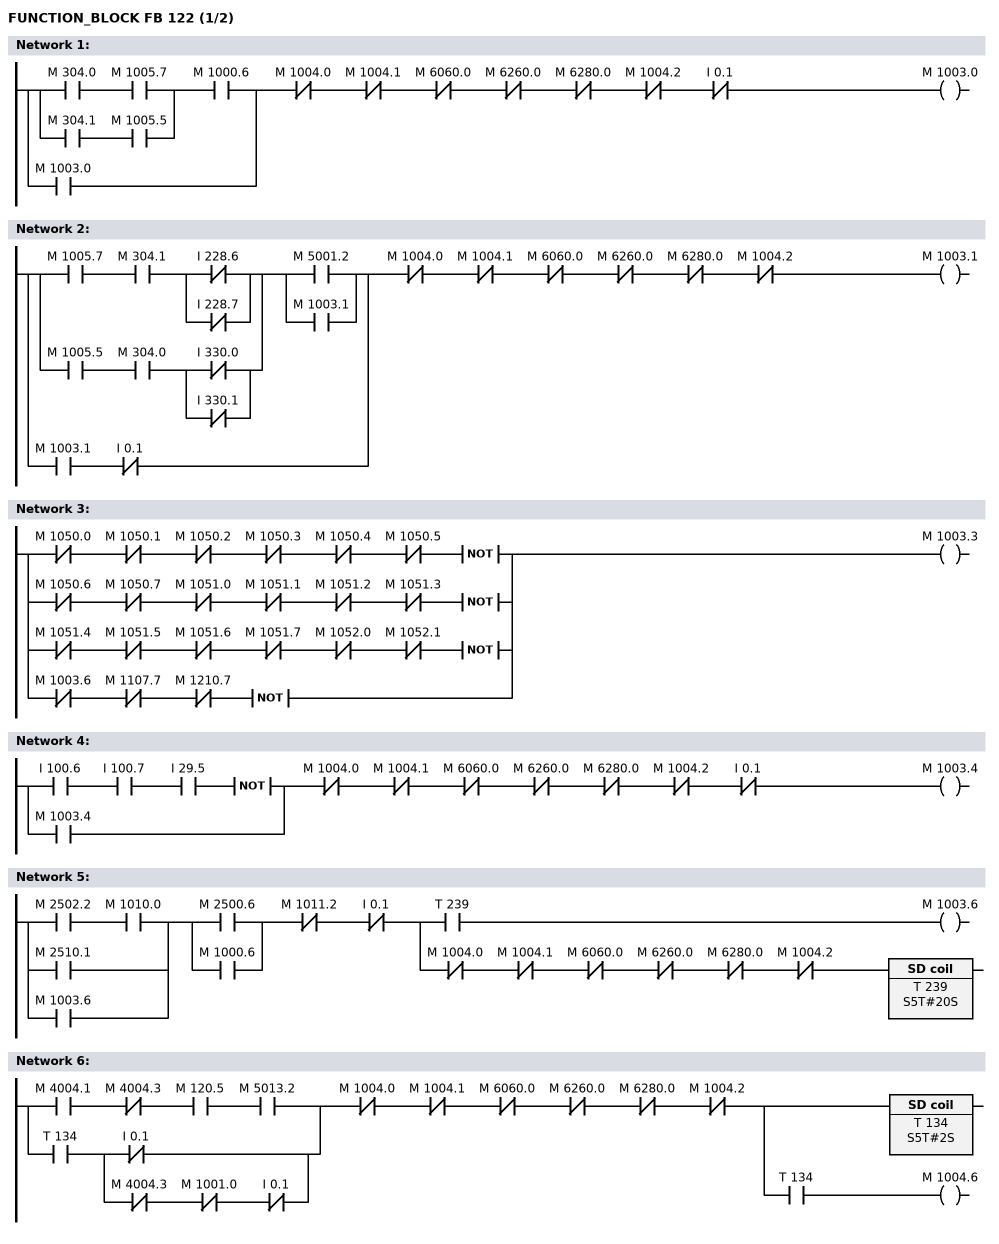

      A(    ;
      A(    ;
      A     M    304.0;
      A     M   1005.7;
      O     ;
      A     M    304.1;
      A     M   1005.5;
      )     ;
      A     M   1000.6;
      O     M   1003.0;
      )     ;
      AN    M   1004.0;
      AN    M   1004.1;
      AN    M   6060.0;
      AN    M   6260.0;
      AN    M   6280.0;
      AN    M   1004.2;
      AN    I      0.1;
      =     M   1003.0;
NETWORK
TITLE =

      A(    ;
      A(    ;
      A     M   1005.7;
      A     M    304.1;
      A(    ;
      ON    I    228.6;
      ON    I    228.7;
      )     ;
      O     ;
      A     M   1005.5;
      A     M    304.0;
      A(    ;
      ON    I    330.0;
      ON    I    330.1;
      )     ;
      )     ;
      A(    ;
      O     M   5001.2;
      O     M   1003.1;
      )     ;
      O     ;
      A     M   1003.1;
      AN    I      0.1;
      )     ;
      AN    M   1004.0;
      AN    M   1004.1;
      AN    M   6060.0;
      AN    M   6260.0;
      AN    M   6280.0;
      AN    M   1004.2;
      =     M   1003.1;
NETWORK
TITLE =

      AN    M   1050.0;
      AN    M   1050.1;
      AN    M   1050.2;
      AN    M   1050.3;
      AN    M   1050.4;
      AN    M   1050.5;
      NOT   ;
      O(    ;
      AN    M   1050.6;
      AN    M   1050.7;
      AN    M   1051.0;
      AN    M   1051.1;
      AN    M   1051.2;
      AN    M   1051.3;
      NOT   ;
      )     ;
      O(    ;
      AN    M   1051.4;
      AN    M   1051.5;
      AN    M   1051.6;
      AN    M   1051.7;
      AN    M   1052.0;
      AN    M   1052.1;
      NOT   ;
      )     ;
      O(    ;
      AN    M   1003.6;
      AN    M   1107.7;
      AN    M   1210.7;
      NOT   ;
      )     ;
      =     M   1003.3;
NETWORK
TITLE =

      A(    ;
      A     I    100.6;
      A     I    100.7;
      A     I     29.5;
      NOT   ;
      O     M   1003.4;
      )     ;
      AN    M   1004.0;
      AN    M   1004.1;
      AN    M   6060.0;
      AN    M   6260.0;
      AN    M   6280.0;
      AN    M   1004.2;
      AN    I      0.1;
      =     M   1003.4;
NETWORK
TITLE =

      A(    ;
      A     M   2502.2;
      A     M   1010.0;
      O     M   2510.1;
      O     M   1003.6;
      )     ;
      A(    ;
      O     M   2500.6;
      O     M   1000.6;
      )     ;
      AN    M   1011.2;
      AN    I      0.1;
      =     L      0.0;
      A     L      0.0;
      A     T    239;
      =     M   1003.6;
      A     L      0.0;
      AN    M   1004.0;
      AN    M   1004.1;
      AN    M   6060.0;
      AN    M   6260.0;
      AN    M   6280.0;
      AN    M   1004.2;
      L     S5T#20S;
      SD    T    239;
NETWORK
TITLE =

      A(    ;
      A     M   4004.1;
      AN    M   4004.3;
      A     M    120.5;
      A     M   5013.2;
      O     ;
      A     T    134;
      A(    ;
      ON    I      0.1;
      O     ;
      AN    M   4004.3;
      AN    M   1001.0;
      AN    I      0.1;
      )     ;
      )     ;
      AN    M   1004.0;
      AN    M   1004.1;
      AN    M   6060.0;
      AN    M   6260.0;
      AN    M   6280.0;
      AN    M   1004.2;
      =     L      0.0;
      A     L      0.0;
      BLD   102;
      L     S5T#2S;
      SD    T    134;
      A     L      0.0;
      A     T    134;
      =     M   1004.6;
NETWORK
TITLE =
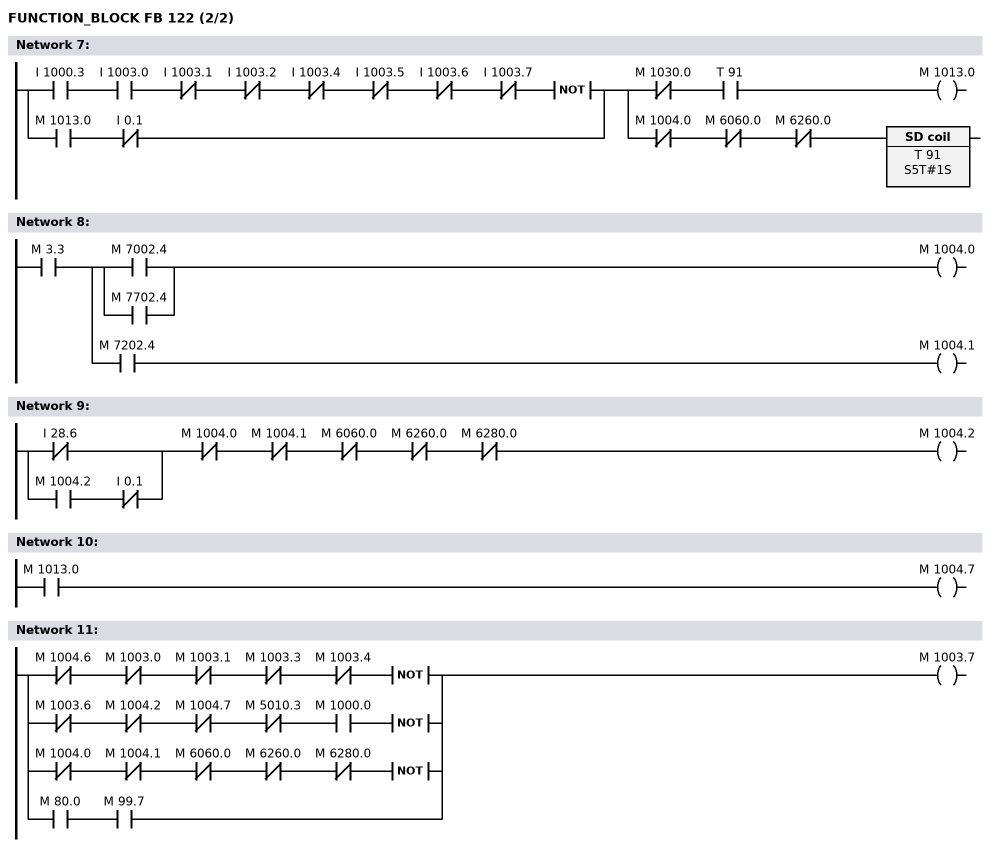

      A     I   1000.3;
      A     I   1003.0;
      AN    I   1003.1;
      AN    I   1003.2;
      AN    I   1003.4;
      AN    I   1003.5;
      AN    I   1003.6;
      AN    I   1003.7;
      NOT   ;
      O     ;
      A     M   1013.0;
      AN    I      0.1;
      =     L      0.0;
      A     L      0.0;
      AN    M   1030.0;
      A     T     91;
      =     M   1013.0;
      A     L      0.0;
      AN    M   1004.0;
      AN    M   6060.0;
      AN    M   6260.0;
      L     S5T#1S;
      SD    T     91;
NETWORK
TITLE =

      A     M      3.3;
      =     L      0.0;
      A     L      0.0;
      A(    ;
      O     M   7002.4;
      O     M   7702.4;
      )     ;
      =     M   1004.0;
      A     L      0.0;
      A     M   7202.4;
      =     M   1004.1;
NETWORK
TITLE =

      A(    ;
      ON    I     28.6;
      O     ;
      A     M   1004.2;
      AN    I      0.1;
      )     ;
      AN    M   1004.0;
      AN    M   1004.1;
      AN    M   6060.0;
      AN    M   6260.0;
      AN    M   6280.0;
      =     M   1004.2;
NETWORK
TITLE =

      A     M   1013.0;
      =     M   1004.7;
NETWORK
TITLE =

      AN    M   1004.6;
      AN    M   1003.0;
      AN    M   1003.1;
      AN    M   1003.3;
      AN    M   1003.4;
      NOT   ;
      O(    ;
      AN    M   1003.6;
      AN    M   1004.2;
      AN    M   1004.7;
      AN    M   5010.3;
      A     M   1000.0;
      NOT   ;
      )     ;
      O(    ;
      AN    M   1004.0;
      AN    M   1004.1;
      AN    M   6060.0;
      AN    M   6260.0;
      AN    M   6280.0;
      NOT   ;
      )     ;
      O     ;
      A     M     80.0;
      A     M     99.7;
      =     M   1003.7;
END_FUNCTION_BLOCK

DATA_BLOCK DB 122
TITLE =
VERSION : 0.0

 FB 122
BEGIN
END_DATA_BLOCK

FUNCTION FC 122 : VOID
TITLE =
VERSION : 0.1

BEGIN
NETWORK
TITLE =

NETWORK
TITLE =
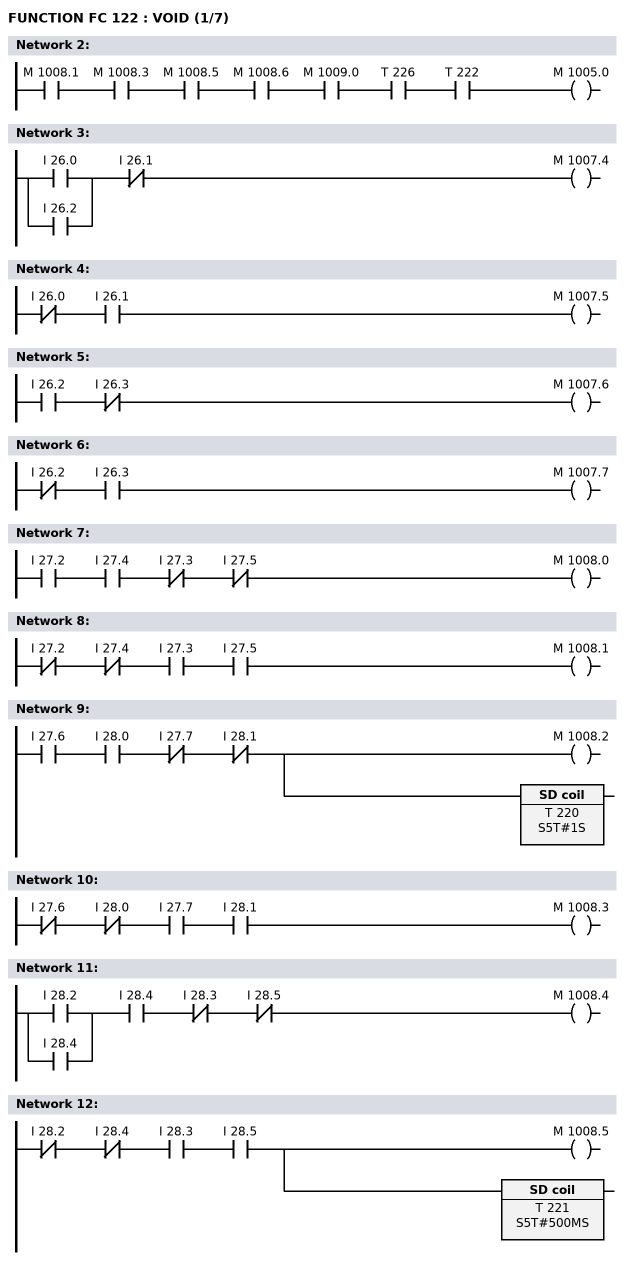

      A     M   1008.1;
      A     M   1008.3;
      A     M   1008.5;
      A     M   1008.6;
      A     M   1009.0;
      A     T    226;
      A     T    222;
      =     M   1005.0;
NETWORK
TITLE =

      A(    ;
      O     I     26.0;
      O     I     26.2;
      )     ;
      AN    I     26.1;
      =     M   1007.4;
NETWORK
TITLE =

      AN    I     26.0;
      A     I     26.1;
      =     M   1007.5;
NETWORK
TITLE =

      A     I     26.2;
      AN    I     26.3;
      =     M   1007.6;
NETWORK
TITLE =

      AN    I     26.2;
      A     I     26.3;
      =     M   1007.7;
NETWORK
TITLE =

      A     I     27.2;
      A     I     27.4;
      AN    I     27.3;
      AN    I     27.5;
      =     M   1008.0;
NETWORK
TITLE =

      AN    I     27.2;
      AN    I     27.4;
      A     I     27.3;
      A     I     27.5;
      =     M   1008.1;
NETWORK
TITLE =

      A     I     27.6;
      A     I     28.0;
      AN    I     27.7;
      AN    I     28.1;
      =     M   1008.2;
      L     S5T#1S;
      SD    T    220;
NETWORK
TITLE =

      AN    I     27.6;
      AN    I     28.0;
      A     I     27.7;
      A     I     28.1;
      =     M   1008.3;
NETWORK
TITLE =

      A(    ;
      O     I     28.2;
      O     I     28.4;
      )     ;
      A     I     28.4;
      AN    I     28.3;
      AN    I     28.5;
      =     M   1008.4;
NETWORK
TITLE =

      AN    I     28.2;
      AN    I     28.4;
      A     I     28.3;
      A     I     28.5;
      =     M   1008.5;
      L     S5T#500MS;
      SD    T    221;
NETWORK
TITLE =
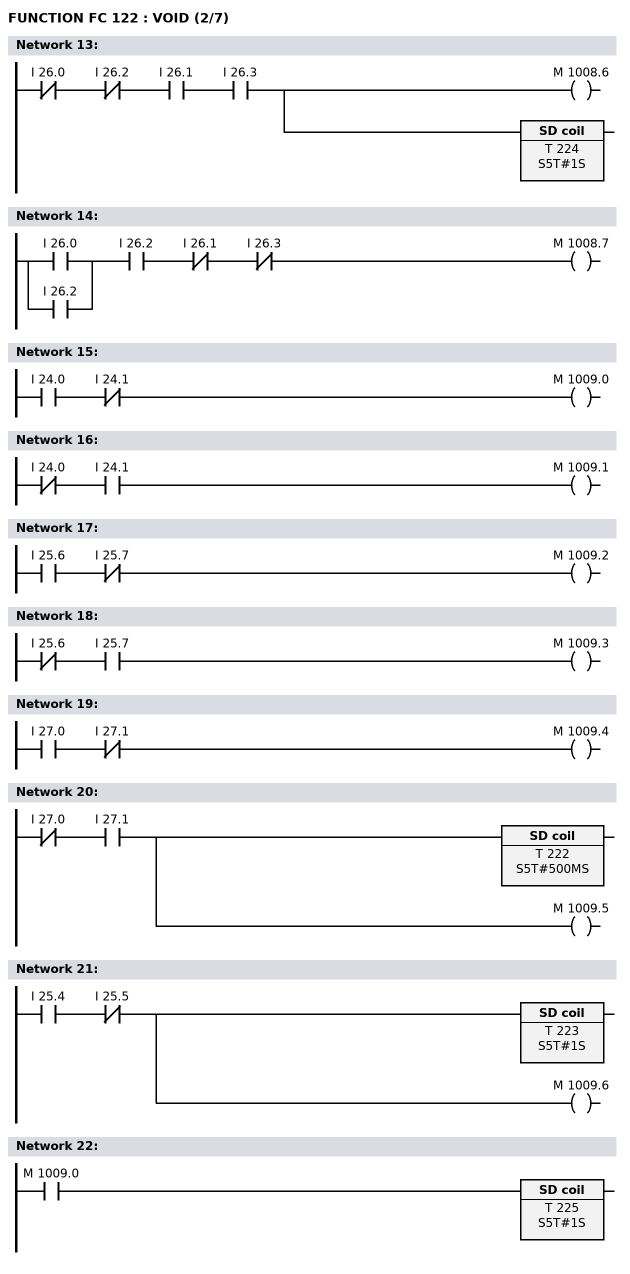

      AN    I     26.0;
      AN    I     26.2;
      A     I     26.1;
      A     I     26.3;
      =     M   1008.6;
      L     S5T#1S;
      SD    T    224;
NETWORK
TITLE =

      A(    ;
      O     I     26.0;
      O     I     26.2;
      )     ;
      A     I     26.2;
      AN    I     26.1;
      AN    I     26.3;
      =     M   1008.7;
NETWORK
TITLE =

      A     I     24.0;
      AN    I     24.1;
      =     M   1009.0;
NETWORK
TITLE =

      AN    I     24.0;
      A     I     24.1;
      =     M   1009.1;
NETWORK
TITLE =

      A     I     25.6;
      AN    I     25.7;
      =     M   1009.2;
NETWORK
TITLE =

      AN    I     25.6;
      A     I     25.7;
      =     M   1009.3;
NETWORK
TITLE =

      A     I     27.0;
      AN    I     27.1;
      =     M   1009.4;
NETWORK
TITLE =

      AN    I     27.0;
      A     I     27.1;
      L     S5T#500MS;
      SD    T    222;
      =     M   1009.5;
NETWORK
TITLE =

      A     I     25.4;
      AN    I     25.5;
      L     S5T#1S;
      SD    T    223;
      =     M   1009.6;
NETWORK
TITLE =

      A     M   1009.0;
      L     S5T#1S;
      SD    T    225;
NETWORK
TITLE =
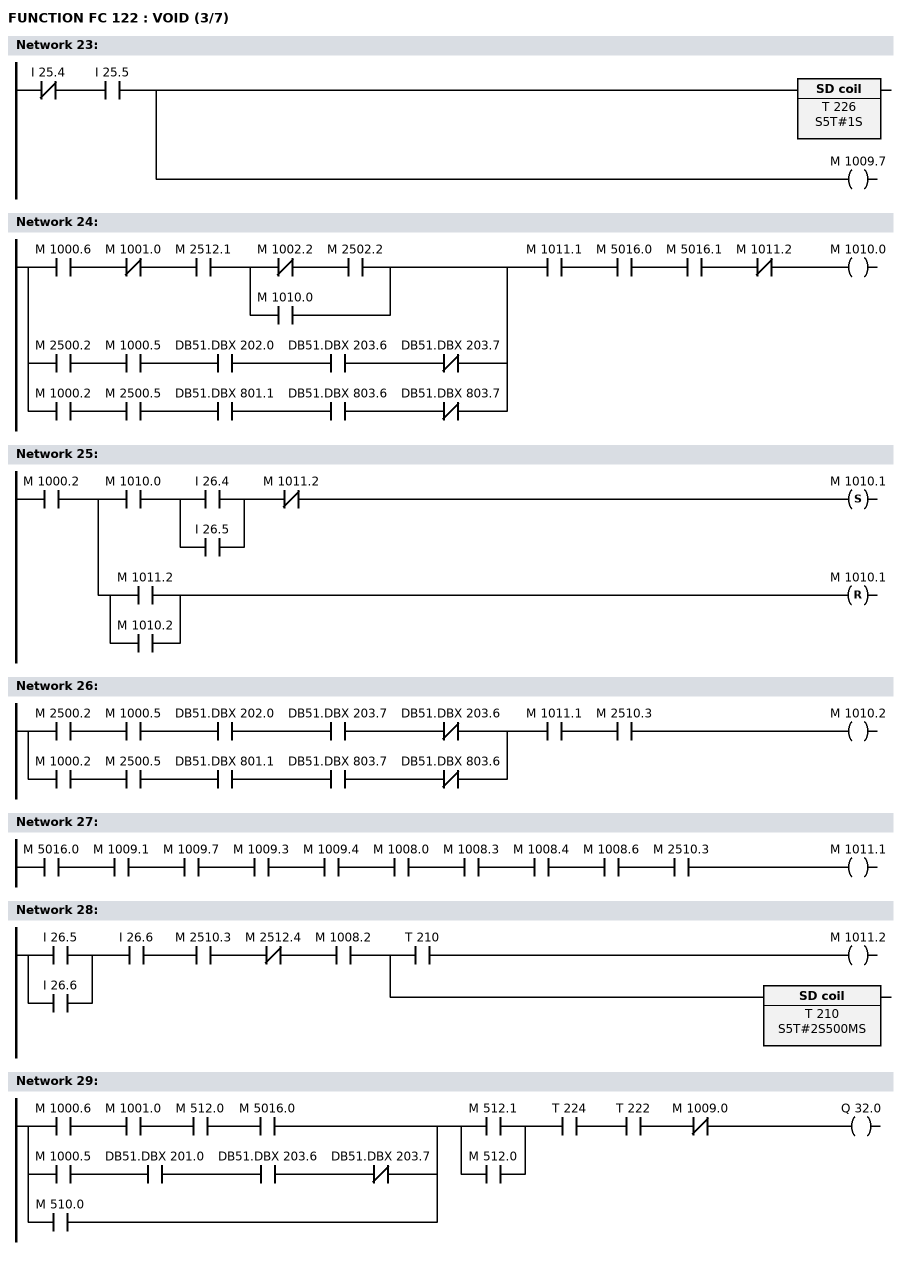

      AN    I     25.4;
      A     I     25.5;
      L     S5T#1S;
      SD    T    226;
      =     M   1009.7;
NETWORK
TITLE =

      A(    ;
      A     M   1000.6;
      AN    M   1001.0;
      A     M   2512.1;
      A(    ;
      AN    M   1002.2;
      A     M   2502.2;
      O     M   1010.0;
      )     ;
      O     ;
      A     M   2500.2;
      A     M   1000.5;
      A     DB51.DBX  202.0;
      A     DB51.DBX  203.6;
      AN    DB51.DBX  203.7;
      O     ;
      A     M   1000.2;
      A     M   2500.5;
      A     DB51.DBX  801.1;
      A     DB51.DBX  803.6;
      AN    DB51.DBX  803.7;
      )     ;
      A     M   1011.1;
      A     M   5016.0;
      A     M   5016.1;
      AN    M   1011.2;
      =     M   1010.0;
NETWORK
TITLE =

      A     M   1000.2;
      =     L      0.0;
      A     L      0.0;
      A     M   1010.0;
      A(    ;
      O     I     26.4;
      O     I     26.5;
      )     ;
      AN    M   1011.2;
      S     M   1010.1;
      A     L      0.0;
      A(    ;
      O     M   1011.2;
      O     M   1010.2;
      )     ;
      R     M   1010.1;
NETWORK
TITLE =

      A(    ;
      A     M   2500.2;
      A     M   1000.5;
      A     DB51.DBX  202.0;
      A     DB51.DBX  203.7;
      AN    DB51.DBX  203.6;
      O     ;
      A     M   1000.2;
      A     M   2500.5;
      A     DB51.DBX  801.1;
      A     DB51.DBX  803.7;
      AN    DB51.DBX  803.6;
      )     ;
      A     M   1011.1;
      A     M   2510.3;
      =     M   1010.2;
NETWORK
TITLE =

      A     M   5016.0;
      A     M   1009.1;
      A     M   1009.7;
      A     M   1009.3;
      A     M   1009.4;
      A     M   1008.0;
      A     M   1008.3;
      A     M   1008.4;
      A     M   1008.6;
      A     M   2510.3;
      =     M   1011.1;
NETWORK
TITLE =

      A(    ;
      O     I     26.5;
      O     I     26.6;
      )     ;
      A     I     26.6;
      A     M   2510.3;
      AN    M   2512.4;
      A     M   1008.2;
      =     L      0.0;
      A     L      0.0;
      A     T    210;
      =     M   1011.2;
      A     L      0.0;
      BLD   102;
      L     S5T#2S500MS;
      SD    T    210;
NETWORK
TITLE =

      A(    ;
      A     M   1000.6;
      A     M   1001.0;
      A     M    512.0;
      A     M   5016.0;
      O     ;
      A     M   1000.5;
      A     DB51.DBX  201.0;
      A     DB51.DBX  203.6;
      AN    DB51.DBX  203.7;
      O     M    510.0;
      )     ;
      A(    ;
      O     M    512.1;
      O     M    512.0;
      )     ;
      A     T    224;
      A     T    222;
      AN    M   1009.0;
      =     Q     32.0;
NETWORK
TITLE =
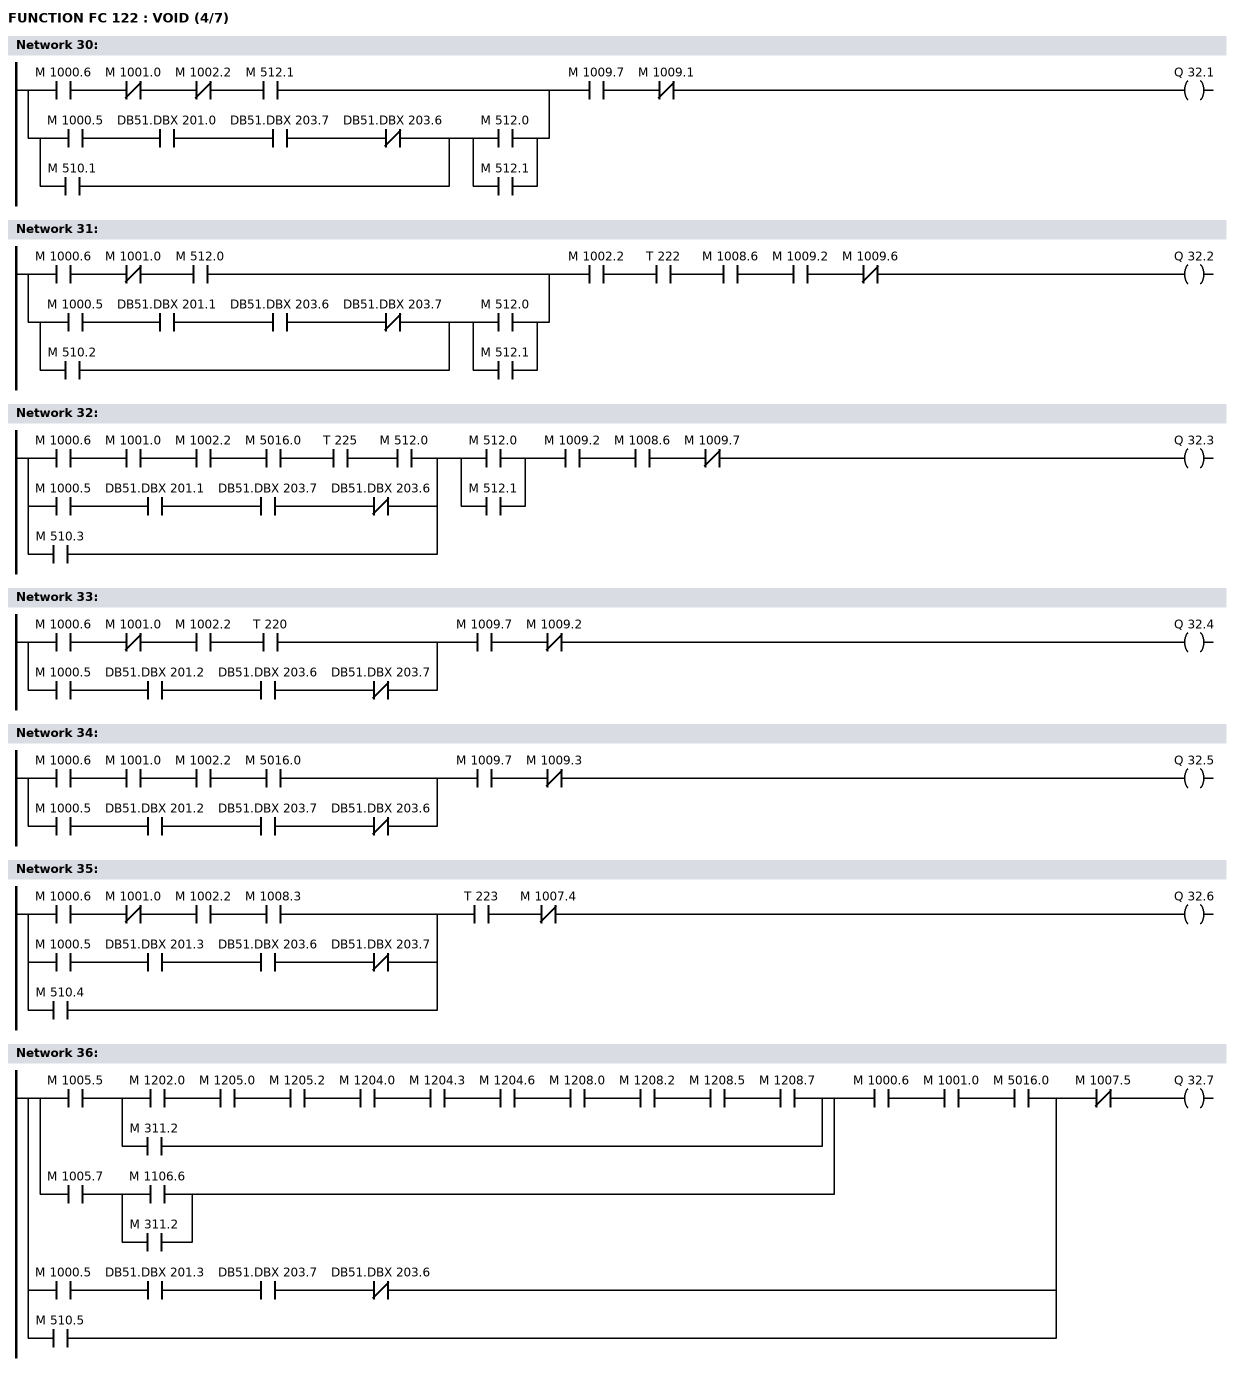

      A(    ;
      A     M   1000.6;
      AN    M   1001.0;
      AN    M   1002.2;
      A     M    512.1;
      O     ;
      A(    ;
      A     M   1000.5;
      A     DB51.DBX  201.0;
      A     DB51.DBX  203.7;
      AN    DB51.DBX  203.6;
      O     M    510.1;
      )     ;
      A(    ;
      O     M    512.0;
      O     M    512.1;
      )     ;
      )     ;
      A     M   1009.7;
      AN    M   1009.1;
      =     Q     32.1;
NETWORK
TITLE =

      A(    ;
      A     M   1000.6;
      AN    M   1001.0;
      A     M    512.0;
      O     ;
      A(    ;
      A     M   1000.5;
      A     DB51.DBX  201.1;
      A     DB51.DBX  203.6;
      AN    DB51.DBX  203.7;
      O     M    510.2;
      )     ;
      A(    ;
      O     M    512.0;
      O     M    512.1;
      )     ;
      )     ;
      A     M   1002.2;
      A     T    222;
      A     M   1008.6;
      A     M   1009.2;
      AN    M   1009.6;
      =     Q     32.2;
NETWORK
TITLE =

      A(    ;
      A     M   1000.6;
      A     M   1001.0;
      A     M   1002.2;
      A     M   5016.0;
      A     T    225;
      A     M    512.0;
      O     ;
      A     M   1000.5;
      A     DB51.DBX  201.1;
      A     DB51.DBX  203.7;
      AN    DB51.DBX  203.6;
      O     M    510.3;
      )     ;
      A(    ;
      O     M    512.0;
      O     M    512.1;
      )     ;
      A     M   1009.2;
      A     M   1008.6;
      AN    M   1009.7;
      =     Q     32.3;
NETWORK
TITLE =

      A(    ;
      A     M   1000.6;
      AN    M   1001.0;
      A     M   1002.2;
      A     T    220;
      O     ;
      A     M   1000.5;
      A     DB51.DBX  201.2;
      A     DB51.DBX  203.6;
      AN    DB51.DBX  203.7;
      )     ;
      A     M   1009.7;
      AN    M   1009.2;
      =     Q     32.4;
NETWORK
TITLE =

      A(    ;
      A     M   1000.6;
      A     M   1001.0;
      A     M   1002.2;
      A     M   5016.0;
      O     ;
      A     M   1000.5;
      A     DB51.DBX  201.2;
      A     DB51.DBX  203.7;
      AN    DB51.DBX  203.6;
      )     ;
      A     M   1009.7;
      AN    M   1009.3;
      =     Q     32.5;
NETWORK
TITLE =

      A(    ;
      A     M   1000.6;
      AN    M   1001.0;
      A     M   1002.2;
      A     M   1008.3;
      O     ;
      A     M   1000.5;
      A     DB51.DBX  201.3;
      A     DB51.DBX  203.6;
      AN    DB51.DBX  203.7;
      O     M    510.4;
      )     ;
      A     T    223;
      AN    M   1007.4;
      =     Q     32.6;
NETWORK
TITLE =

      A(    ;
      A(    ;
      A     M   1005.5;
      A(    ;
      A     M   1202.0;
      A     M   1205.0;
      A     M   1205.2;
      A     M   1204.0;
      A     M   1204.3;
      A     M   1204.6;
      A     M   1208.0;
      A     M   1208.2;
      A     M   1208.5;
      A     M   1208.7;
      O     M    311.2;
      )     ;
      O     ;
      A     M   1005.7;
      A(    ;
      O     M   1106.6;
      O     M    311.2;
      )     ;
      )     ;
      A     M   1000.6;
      A     M   1001.0;
      A     M   5016.0;
      O     ;
      A     M   1000.5;
      A     DB51.DBX  201.3;
      A     DB51.DBX  203.7;
      AN    DB51.DBX  203.6;
      O     M    510.5;
      )     ;
      AN    M   1007.5;
      =     Q     32.7;
NETWORK
TITLE =
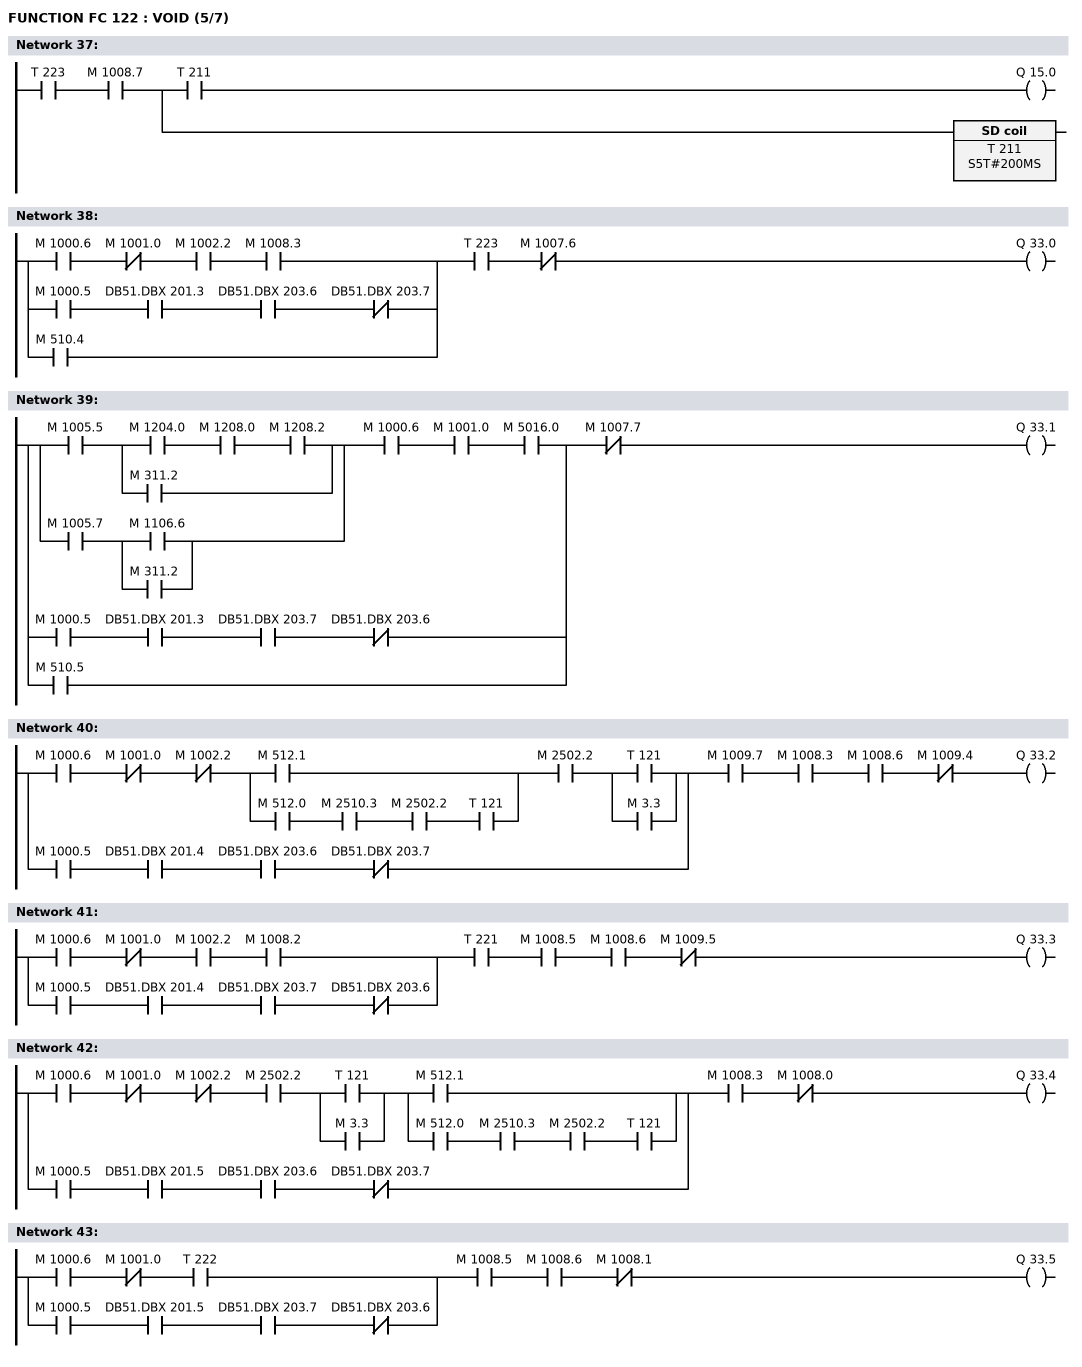

      A     T    223;
      A     M   1008.7;
      =     L      0.0;
      A     L      0.0;
      A     T    211;
      =     Q     15.0;
      A     L      0.0;
      BLD   102;
      L     S5T#200MS;
      SD    T    211;
NETWORK
TITLE =

      A(    ;
      A     M   1000.6;
      AN    M   1001.0;
      A     M   1002.2;
      A     M   1008.3;
      O     ;
      A     M   1000.5;
      A     DB51.DBX  201.3;
      A     DB51.DBX  203.6;
      AN    DB51.DBX  203.7;
      O     M    510.4;
      )     ;
      A     T    223;
      AN    M   1007.6;
      =     Q     33.0;
NETWORK
TITLE =

      A(    ;
      A(    ;
      A     M   1005.5;
      A(    ;
      A     M   1204.0;
      A     M   1208.0;
      A     M   1208.2;
      O     M    311.2;
      )     ;
      O     ;
      A     M   1005.7;
      A(    ;
      O     M   1106.6;
      O     M    311.2;
      )     ;
      )     ;
      A     M   1000.6;
      A     M   1001.0;
      A     M   5016.0;
      O     ;
      A     M   1000.5;
      A     DB51.DBX  201.3;
      A     DB51.DBX  203.7;
      AN    DB51.DBX  203.6;
      O     M    510.5;
      )     ;
      AN    M   1007.7;
      =     Q     33.1;
NETWORK
TITLE =

      A(    ;
      A     M   1000.6;
      AN    M   1001.0;
      AN    M   1002.2;
      A(    ;
      O     M    512.1;
      O     ;
      A     M    512.0;
      A     M   2510.3;
      A     M   2502.2;
      A     T    121;
      )     ;
      A     M   2502.2;
      A(    ;
      O     T    121;
      O     M      3.3;
      )     ;
      O     ;
      A     M   1000.5;
      A     DB51.DBX  201.4;
      A     DB51.DBX  203.6;
      AN    DB51.DBX  203.7;
      )     ;
      A     M   1009.7;
      A     M   1008.3;
      A     M   1008.6;
      AN    M   1009.4;
      =     Q     33.2;
NETWORK
TITLE =

      A(    ;
      A     M   1000.6;
      AN    M   1001.0;
      A     M   1002.2;
      A     M   1008.2;
      O     ;
      A     M   1000.5;
      A     DB51.DBX  201.4;
      A     DB51.DBX  203.7;
      AN    DB51.DBX  203.6;
      )     ;
      A     T    221;
      A     M   1008.5;
      A     M   1008.6;
      AN    M   1009.5;
      =     Q     33.3;
NETWORK
TITLE =

      A(    ;
      A     M   1000.6;
      AN    M   1001.0;
      AN    M   1002.2;
      A     M   2502.2;
      A(    ;
      O     T    121;
      O     M      3.3;
      )     ;
      A(    ;
      O     M    512.1;
      O     ;
      A     M    512.0;
      A     M   2510.3;
      A     M   2502.2;
      A     T    121;
      )     ;
      O     ;
      A     M   1000.5;
      A     DB51.DBX  201.5;
      A     DB51.DBX  203.6;
      AN    DB51.DBX  203.7;
      )     ;
      A     M   1008.3;
      AN    M   1008.0;
      =     Q     33.4;
NETWORK
TITLE =

      A(    ;
      A     M   1000.6;
      AN    M   1001.0;
      A     T    222;
      O     ;
      A     M   1000.5;
      A     DB51.DBX  201.5;
      A     DB51.DBX  203.7;
      AN    DB51.DBX  203.6;
      )     ;
      A     M   1008.5;
      A     M   1008.6;
      AN    M   1008.1;
      =     Q     33.5;
NETWORK
TITLE =
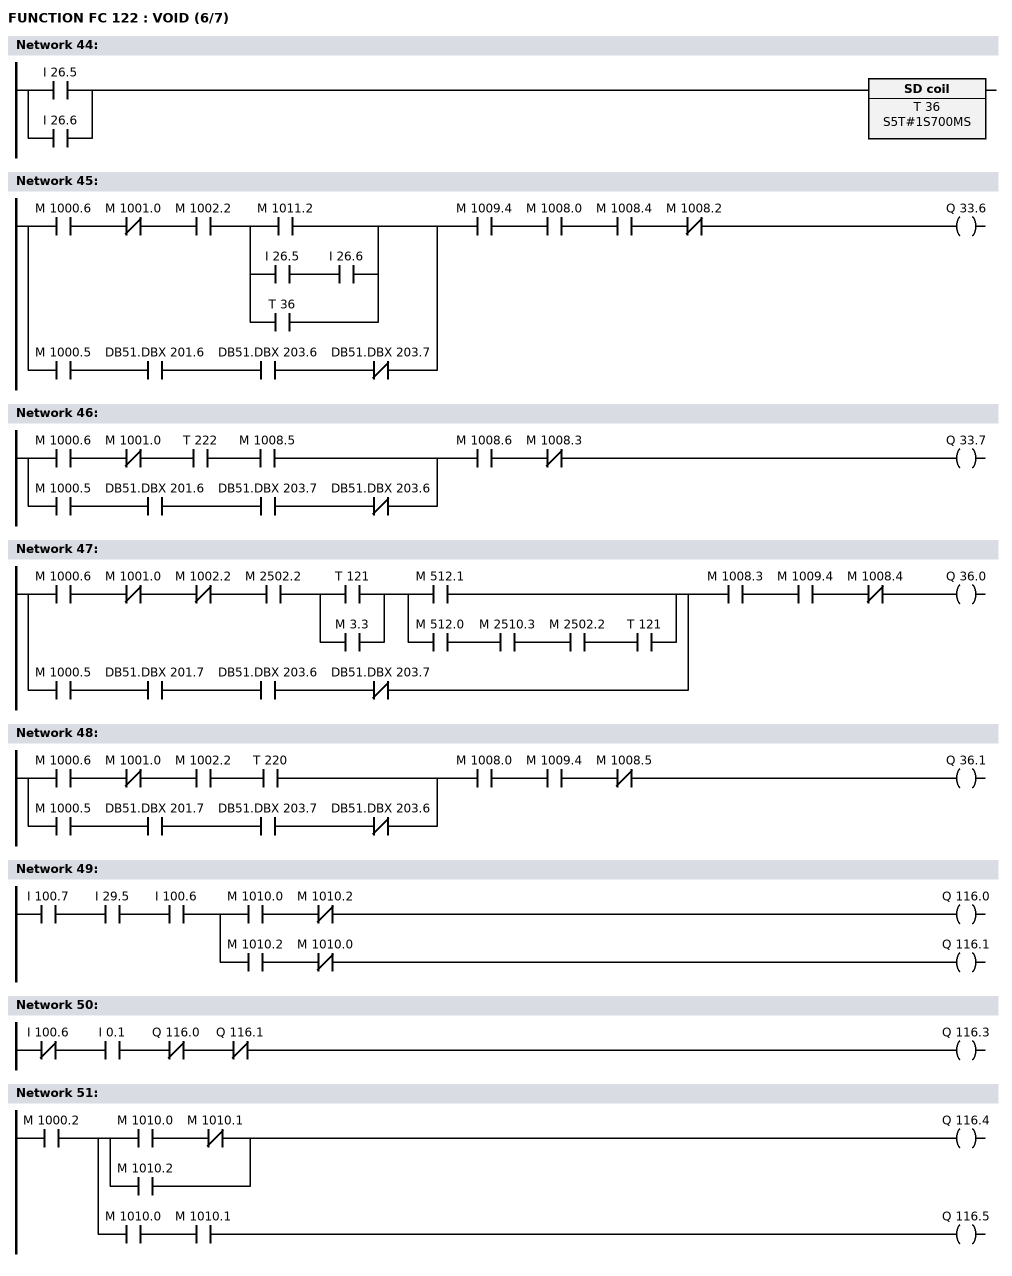

      O     I     26.5;
      O     I     26.6;
      L     S5T#1S700MS;
      SD    T     36;
NETWORK
TITLE =

      A(    ;
      A     M   1000.6;
      AN    M   1001.0;
      A     M   1002.2;
      A(    ;
      O     M   1011.2;
      O     ;
      A     I     26.5;
      A     I     26.6;
      O     T     36;
      )     ;
      O     ;
      A     M   1000.5;
      A     DB51.DBX  201.6;
      A     DB51.DBX  203.6;
      AN    DB51.DBX  203.7;
      )     ;
      A     M   1009.4;
      A     M   1008.0;
      A     M   1008.4;
      AN    M   1008.2;
      =     Q     33.6;
NETWORK
TITLE =

      A(    ;
      A     M   1000.6;
      AN    M   1001.0;
      A     T    222;
      A     M   1008.5;
      O     ;
      A     M   1000.5;
      A     DB51.DBX  201.6;
      A     DB51.DBX  203.7;
      AN    DB51.DBX  203.6;
      )     ;
      A     M   1008.6;
      AN    M   1008.3;
      =     Q     33.7;
NETWORK
TITLE =

      A(    ;
      A     M   1000.6;
      AN    M   1001.0;
      AN    M   1002.2;
      A     M   2502.2;
      A(    ;
      O     T    121;
      O     M      3.3;
      )     ;
      A(    ;
      O     M    512.1;
      O     ;
      A     M    512.0;
      A     M   2510.3;
      A     M   2502.2;
      A     T    121;
      )     ;
      O     ;
      A     M   1000.5;
      A     DB51.DBX  201.7;
      A     DB51.DBX  203.6;
      AN    DB51.DBX  203.7;
      )     ;
      A     M   1008.3;
      A     M   1009.4;
      AN    M   1008.4;
      =     Q     36.0;
NETWORK
TITLE =

      A(    ;
      A     M   1000.6;
      AN    M   1001.0;
      A     M   1002.2;
      A     T    220;
      O     ;
      A     M   1000.5;
      A     DB51.DBX  201.7;
      A     DB51.DBX  203.7;
      AN    DB51.DBX  203.6;
      )     ;
      A     M   1008.0;
      A     M   1009.4;
      AN    M   1008.5;
      =     Q     36.1;
NETWORK
TITLE =

      A     I    100.7;
      A     I     29.5;
      A     I    100.6;
      =     L      0.0;
      A     L      0.0;
      A     M   1010.0;
      AN    M   1010.2;
      =     Q    116.0;
      A     L      0.0;
      A     M   1010.2;
      AN    M   1010.0;
      =     Q    116.1;
NETWORK
TITLE =

      AN    I    100.6;
      A     I      0.1;
      AN    Q    116.0;
      AN    Q    116.1;
      =     Q    116.3;
NETWORK
TITLE =

      A     M   1000.2;
      =     L      0.0;
      A     L      0.0;
      A(    ;
      A     M   1010.0;
      AN    M   1010.1;
      O     M   1010.2;
      )     ;
      =     Q    116.4;
      A     L      0.0;
      A     M   1010.0;
      A     M   1010.1;
      =     Q    116.5;
NETWORK
TITLE =
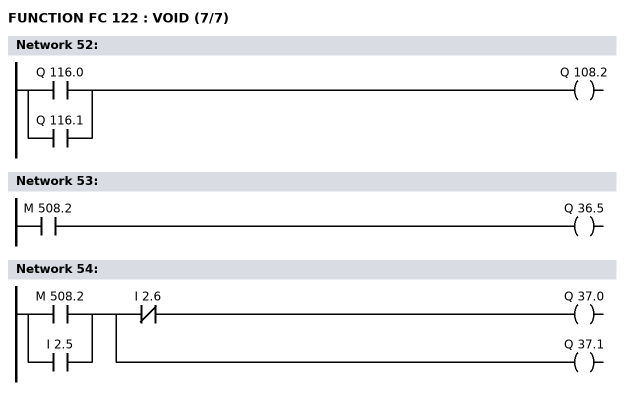

      O     Q    116.0;
      O     Q    116.1;
      =     Q    108.2;
NETWORK
TITLE =

      A     M    508.2;
      =     Q     36.5;
NETWORK
TITLE =

      O     M    508.2;
      O     I      2.5;
      =     L      0.0;
      A     L      0.0;
      AN    I      2.6;
      =     Q     37.0;
      A     L      0.0;
      BLD   102;
      =     Q     37.1;
END_FUNCTION

FUNCTION_BLOCK FB 123
TITLE =
VERSION : 0.1


VAR
  S702_LM_DC_PIN : FB 424;
  S702_LM_DC_1ST_CLAMP1 : FB 424;
  S702_LM_DC_1ST_CLAMP2 : FB 424;
  S702_LM_DC_1ST_CLAMP3 : FB 424;
  S702_LM_DC_1ST_CLAMP4 : FB 424;
  S702_LM_DC_2ND_CLAMP1 : FB 424;
  S702_LM_DC_2ND_CLAMP2 : FB 424;
  S702_LM_DC_2ND_CLAMP3 : FB 424;
  S702_LM_DC_2ND_CLAMP4 : FB 424;
  S702_LM_DC_2ND_CLAMP5 : FB 424;
  S702_LM_DC_STK_PIN : FB 424;
  S702_LM_DC_OTR_CLAMP : FB 424;
  S702_LM_DC_ASSY_CLAMP : FB 424;
  S702_LM_DC_FF_PIN : FB 424;
  S702_LM_DC_FF_CLAMP : FB 424;
  S702_LM_DC_2ND_CLAMP6 : FB 424;
  S702_LM_DC_2ND_CLAMP7 : FB 424;
  S702_LM_DC_1ST_CLAMP5 : FB 424;
END_VAR
BEGIN
NETWORK
TITLE =
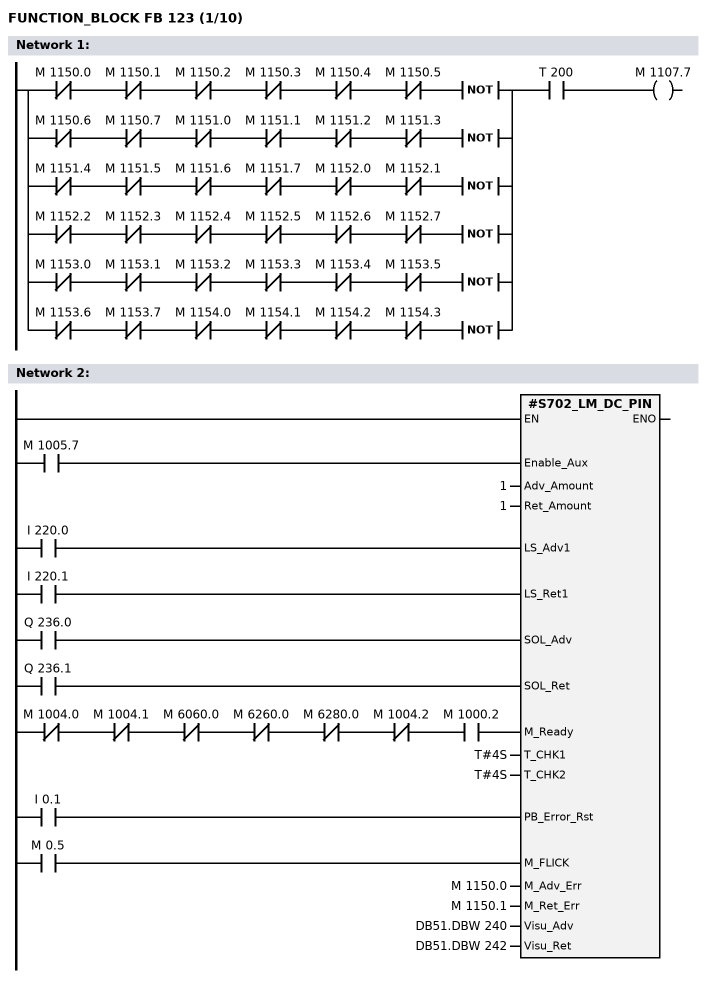

      A(    ;
      AN    M   1150.0;
      AN    M   1150.1;
      AN    M   1150.2;
      AN    M   1150.3;
      AN    M   1150.4;
      AN    M   1150.5;
      NOT   ;
      O(    ;
      AN    M   1150.6;
      AN    M   1150.7;
      AN    M   1151.0;
      AN    M   1151.1;
      AN    M   1151.2;
      AN    M   1151.3;
      NOT   ;
      )     ;
      O(    ;
      AN    M   1151.4;
      AN    M   1151.5;
      AN    M   1151.6;
      AN    M   1151.7;
      AN    M   1152.0;
      AN    M   1152.1;
      NOT   ;
      )     ;
      O(    ;
      AN    M   1152.2;
      AN    M   1152.3;
      AN    M   1152.4;
      AN    M   1152.5;
      AN    M   1152.6;
      AN    M   1152.7;
      NOT   ;
      )     ;
      O(    ;
      AN    M   1153.0;
      AN    M   1153.1;
      AN    M   1153.2;
      AN    M   1153.3;
      AN    M   1153.4;
      AN    M   1153.5;
      NOT   ;
      )     ;
      O(    ;
      AN    M   1153.6;
      AN    M   1153.7;
      AN    M   1154.0;
      AN    M   1154.1;
      AN    M   1154.2;
      AN    M   1154.3;
      NOT   ;
      )     ;
      )     ;
      A     T    200;
      =     M   1107.7;
NETWORK
TITLE =

      A     M   1005.7;
      =     L      0.0;
      BLD   103;
      A     I    220.0;
      =     L      0.1;
      BLD   103;
      A     I    220.1;
      =     L      0.2;
      BLD   103;
      A     Q    236.0;
      =     L      1.1;
      BLD   103;
      A     Q    236.1;
      =     L      1.2;
      BLD   103;
      AN    M   1004.0;
      AN    M   1004.1;
      AN    M   6060.0;
      AN    M   6260.0;
      AN    M   6280.0;
      AN    M   1004.2;
      A     M   1000.2;
      =     L      1.3;
      BLD   103;
      A     I      0.1;
      =     L      1.5;
      BLD   103;
      A     M      0.5;
      =     L      1.6;
      BLD   103;
      CALL #S702_LM_DC_PIN (
           Enable_Aux               := L      0.0,
           Adv_Amount               := 1,
           Ret_Amount               := 1,
           LS_Adv1                  := L      0.1,
           LS_Ret1                  := L      0.2,
           SOL_Adv                  := L      1.1,
           SOL_Ret                  := L      1.2,
           M_Ready                  := L      1.3,
           T_CHK1                   := T#4S,
           T_CHK2                   := T#4S,
           PB_Error_Rst             := L      1.5,
           M_FLICK                  := L      1.6,
           M_Adv_Err                := M   1150.0,
           M_Ret_Err                := M   1150.1,
           Visu_Adv                 := DB51.DBW  240,
           Visu_Ret                 := DB51.DBW  242);
      NOP   0;
NETWORK
TITLE =
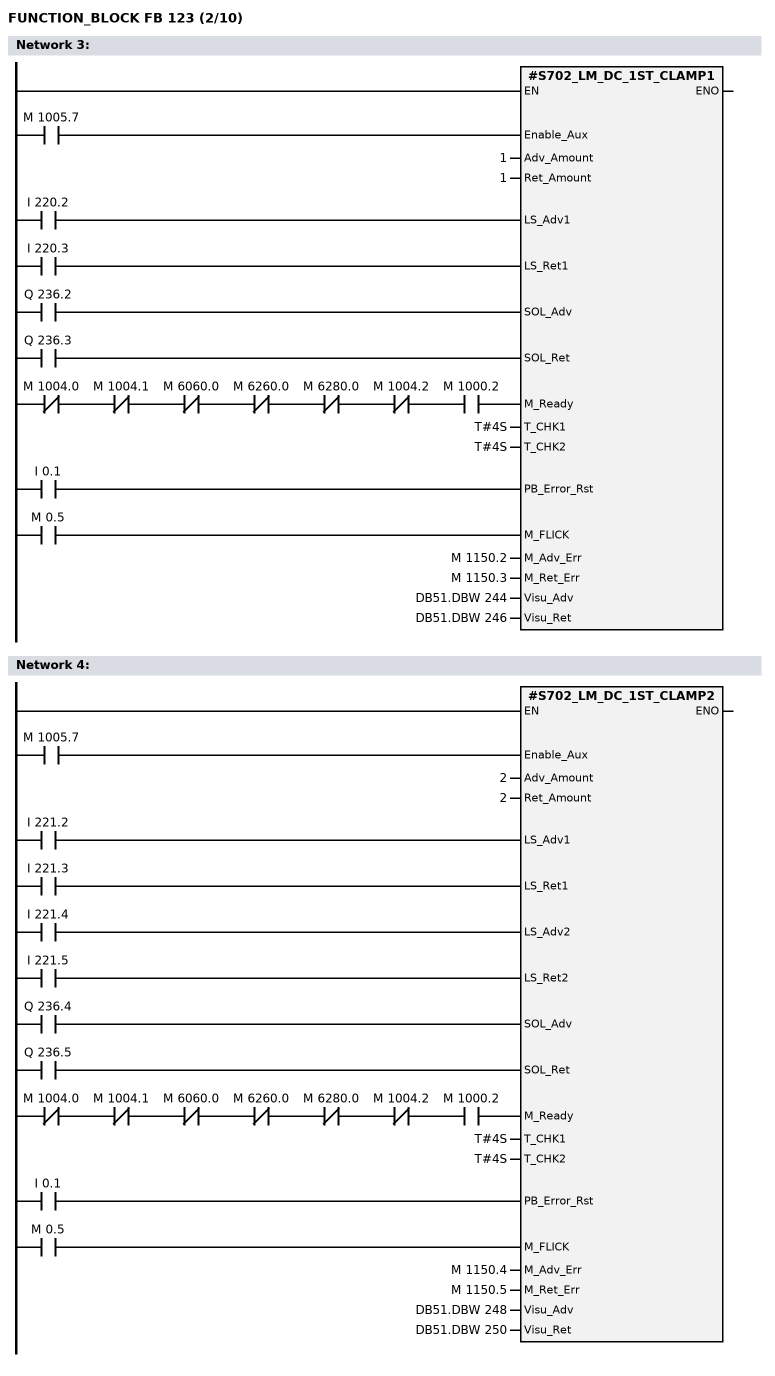

      A     M   1005.7;
      =     L      0.0;
      BLD   103;
      A     I    220.2;
      =     L      0.1;
      BLD   103;
      A     I    220.3;
      =     L      0.2;
      BLD   103;
      A     Q    236.2;
      =     L      1.1;
      BLD   103;
      A     Q    236.3;
      =     L      1.2;
      BLD   103;
      AN    M   1004.0;
      AN    M   1004.1;
      AN    M   6060.0;
      AN    M   6260.0;
      AN    M   6280.0;
      AN    M   1004.2;
      A     M   1000.2;
      =     L      1.3;
      BLD   103;
      A     I      0.1;
      =     L      1.5;
      BLD   103;
      A     M      0.5;
      =     L      1.6;
      BLD   103;
      CALL #S702_LM_DC_1ST_CLAMP1 (
           Enable_Aux               := L      0.0,
           Adv_Amount               := 1,
           Ret_Amount               := 1,
           LS_Adv1                  := L      0.1,
           LS_Ret1                  := L      0.2,
           SOL_Adv                  := L      1.1,
           SOL_Ret                  := L      1.2,
           M_Ready                  := L      1.3,
           T_CHK1                   := T#4S,
           T_CHK2                   := T#4S,
           PB_Error_Rst             := L      1.5,
           M_FLICK                  := L      1.6,
           M_Adv_Err                := M   1150.2,
           M_Ret_Err                := M   1150.3,
           Visu_Adv                 := DB51.DBW  244,
           Visu_Ret                 := DB51.DBW  246);
      NOP   0;
NETWORK
TITLE =

      A     M   1005.7;
      =     L      0.0;
      BLD   103;
      A     I    221.2;
      =     L      0.1;
      BLD   103;
      A     I    221.3;
      =     L      0.2;
      BLD   103;
      A     I    221.4;
      =     L      0.3;
      BLD   103;
      A     I    221.5;
      =     L      0.4;
      BLD   103;
      A     Q    236.4;
      =     L      1.1;
      BLD   103;
      A     Q    236.5;
      =     L      1.2;
      BLD   103;
      AN    M   1004.0;
      AN    M   1004.1;
      AN    M   6060.0;
      AN    M   6260.0;
      AN    M   6280.0;
      AN    M   1004.2;
      A     M   1000.2;
      =     L      1.3;
      BLD   103;
      A     I      0.1;
      =     L      1.5;
      BLD   103;
      A     M      0.5;
      =     L      1.6;
      BLD   103;
      CALL #S702_LM_DC_1ST_CLAMP2 (
           Enable_Aux               := L      0.0,
           Adv_Amount               := 2,
           Ret_Amount               := 2,
           LS_Adv1                  := L      0.1,
           LS_Ret1                  := L      0.2,
           LS_Adv2                  := L      0.3,
           LS_Ret2                  := L      0.4,
           SOL_Adv                  := L      1.1,
           SOL_Ret                  := L      1.2,
           M_Ready                  := L      1.3,
           T_CHK1                   := T#4S,
           T_CHK2                   := T#4S,
           PB_Error_Rst             := L      1.5,
           M_FLICK                  := L      1.6,
           M_Adv_Err                := M   1150.4,
           M_Ret_Err                := M   1150.5,
           Visu_Adv                 := DB51.DBW  248,
           Visu_Ret                 := DB51.DBW  250);
      NOP   0;
NETWORK
TITLE =
